   1:  PR[GP1:91,3] = PR[GP1:90,3] + 60.500;
   1:L PR[91] 10mm/sec CNT100;
   1:  PR[GP1:91,1] = PR[GP1:90,1] + -5.194;
   1:  PR[GP1:91,2] = PR[GP1:90,2] + -19.396;
   1:L PR[91] 10mm/sec CNT100;
   1:  PR[GP1:91,1] = PR[GP1:90,1] + -4.305;
   1:  PR[GP1:91,2] = PR[GP1:90,2] + -20.285;
   1:L PR[91] 10mm/sec CNT100;
   1:  PR[GP1:91,1] = PR[GP1:90,1] + -1.571;
   1:  PR[GP1:91,2] = PR[GP1:90,2] + -23.234;
   1:L PR[91] 10mm/sec CNT100;
   1:  PR[GP1:91,1] = PR[GP1:90,1] + -0.513;
   1:  PR[GP1:91,2] = PR[GP1:90,2] + -24.061;
   1:L PR[91] 10mm/sec CNT100;
   1:  PR[GP1:91,1] = PR[GP1:90,1] + 2.835;
   1:  PR[GP1:91,2] = PR[GP1:90,2] + -26.549;
   1:L PR[91] 10mm/sec CNT100;
   1:  PR[GP1:91,1] = PR[GP1:90,1] + 5.911;
   1:  PR[GP1:91,2] = PR[GP1:90,2] + -28.205;
   1:L PR[91] 10mm/sec CNT100;
   1:  PR[GP1:91,1] = PR[GP1:90,1] + 7.682;
   1:  PR[GP1:91,2] = PR[GP1:90,2] + -29.088;
   1:L PR[91] 10mm/sec CNT100;
   1:  PR[GP1:91,1] = PR[GP1:90,1] + 12.488;
   1:  PR[GP1:91,2] = PR[GP1:90,2] + -30.711;
   1:L PR[91] 10mm/sec CNT100;
   1:  PR[GP1:91,1] = PR[GP1:90,1] + 12.831;
   1:  PR[GP1:91,2] = PR[GP1:90,2] + -30.841;
   1:L PR[91] 10mm/sec CNT100;
   1:  PR[GP1:91,1] = PR[GP1:90,1] + 18.234;
   1:  PR[GP1:91,2] = PR[GP1:90,2] + -31.928;
   1:L PR[91] 10mm/sec CNT100;
   1:  PR[GP1:91,1] = PR[GP1:90,1] + 19.560;
   1:  PR[GP1:91,2] = PR[GP1:90,2] + -32.004;
   1:L PR[91] 10mm/sec CNT100;
   1:  PR[GP1:91,1] = PR[GP1:90,1] + 22.620;
   1:  PR[GP1:91,2] = PR[GP1:90,2] + -32.037;
   1:L PR[91] 10mm/sec CNT100;
   1:  PR[GP1:91,1] = PR[GP1:90,1] + 24.592;
   1:  PR[GP1:91,2] = PR[GP1:90,2] + -31.874;
   1:L PR[91] 10mm/sec CNT100;
   1:  PR[GP1:91,1] = PR[GP1:90,1] + 25.073;
   1:  PR[GP1:91,2] = PR[GP1:90,2] + -31.805;
   1:L PR[91] 10mm/sec CNT100;
   1:  PR[GP1:91,1] = PR[GP1:90,1] + 25.618;
   1:  PR[GP1:91,2] = PR[GP1:90,2] + -31.695;
   1:L PR[91] 10mm/sec CNT100;
   1:  PR[GP1:91,1] = PR[GP1:90,1] + 27.898;
   1:  PR[GP1:91,2] = PR[GP1:90,2] + -31.148;
   1:L PR[91] 10mm/sec CNT100;
   1:  PR[GP1:91,1] = PR[GP1:90,1] + 28.378;
   1:  PR[GP1:91,2] = PR[GP1:90,2] + -31.011;
   1:L PR[91] 10mm/sec CNT100;
   1:  PR[GP1:91,1] = PR[GP1:90,1] + 31.208;
   1:  PR[GP1:91,2] = PR[GP1:90,2] + -29.808;
   1:L PR[91] 10mm/sec CNT100;
   1:  PR[GP1:91,1] = PR[GP1:90,1] + 31.485;
   1:  PR[GP1:91,2] = PR[GP1:90,2] + -29.654;
   1:L PR[91] 10mm/sec CNT100;
   1:  PR[GP1:91,1] = PR[GP1:90,1] + 33.797;
   1:  PR[GP1:91,2] = PR[GP1:90,2] + -28.079;
   1:L PR[91] 10mm/sec CNT100;
   1:  PR[GP1:91,1] = PR[GP1:90,1] + 33.896;
   1:  PR[GP1:91,2] = PR[GP1:90,2] + -28.003;
   1:L PR[91] 10mm/sec CNT100;
   1:  PR[GP1:91,1] = PR[GP1:90,1] + 35.916;
   1:  PR[GP1:91,2] = PR[GP1:90,2] + -25.895;
   1:L PR[91] 10mm/sec CNT100;
   1:  PR[GP1:91,1] = PR[GP1:90,1] + 37.425;
   1:  PR[GP1:91,2] = PR[GP1:90,2] + -23.399;
   1:L PR[91] 10mm/sec CNT100;
   1:  PR[GP1:91,1] = PR[GP1:90,1] + 38.343;
   1:  PR[GP1:91,2] = PR[GP1:90,2] + -20.620;
   1:L PR[91] 10mm/sec CNT100;
   1:  PR[GP1:91,1] = PR[GP1:90,1] + 38.648;
   1:  PR[GP1:91,2] = PR[GP1:90,2] + -17.822;
   1:L PR[91] 10mm/sec CNT100;
   1:  PR[GP1:91,1] = PR[GP1:90,1] + 38.658;
   1:  PR[GP1:91,2] = PR[GP1:90,2] + -17.576;
   1:L PR[91] 10mm/sec CNT100;
   1:  PR[GP1:91,1] = PR[GP1:90,1] + 38.397;
   1:  PR[GP1:91,2] = PR[GP1:90,2] + -14.692;
   1:L PR[91] 10mm/sec CNT100;
   1:  PR[GP1:91,1] = PR[GP1:90,1] + 38.333;
   1:  PR[GP1:91,2] = PR[GP1:90,2] + -14.338;
   1:L PR[91] 10mm/sec CNT100;
   1:  PR[GP1:91,1] = PR[GP1:90,1] + 38.245;
   1:  PR[GP1:91,2] = PR[GP1:90,2] + -13.997;
   1:L PR[91] 10mm/sec CNT100;
   1:  PR[GP1:91,1] = PR[GP1:90,1] + 37.589;
   1:  PR[GP1:91,2] = PR[GP1:90,2] + -11.656;
   1:L PR[91] 10mm/sec CNT100;
   1:  PR[GP1:91,1] = PR[GP1:90,1] + 37.155;
   1:  PR[GP1:91,2] = PR[GP1:90,2] + -10.549;
   1:L PR[91] 10mm/sec CNT100;
   1:  PR[GP1:91,1] = PR[GP1:90,1] + 36.548;
   1:  PR[GP1:91,2] = PR[GP1:90,2] + -9.179;
   1:L PR[91] 10mm/sec CNT100;
   1:  PR[GP1:91,1] = PR[GP1:90,1] + 36.145;
   1:  PR[GP1:91,2] = PR[GP1:90,2] + -8.389;
   1:L PR[91] 10mm/sec CNT100;
   1:  PR[GP1:91,1] = PR[GP1:90,1] + 34.970;
   1:  PR[GP1:91,2] = PR[GP1:90,2] + -6.423;
   1:L PR[91] 10mm/sec CNT100;
   1:  PR[GP1:91,1] = PR[GP1:90,1] + 34.010;
   1:  PR[GP1:91,2] = PR[GP1:90,2] + -5.069;
   1:L PR[91] 10mm/sec CNT100;
   1:  PR[GP1:91,1] = PR[GP1:90,1] + 33.678;
   1:  PR[GP1:91,2] = PR[GP1:90,2] + -4.630;
   1:L PR[91] 10mm/sec CNT100;
   1:  PR[GP1:91,1] = PR[GP1:90,1] + 32.304;
   1:  PR[GP1:91,2] = PR[GP1:90,2] + -2.989;
   1:L PR[91] 10mm/sec CNT100;
   1:  PR[GP1:91,1] = PR[GP1:90,1] + 31.898;
   1:  PR[GP1:91,2] = PR[GP1:90,2] + -2.568;
   1:L PR[91] 10mm/sec CNT100;
   1:  PR[GP1:91,1] = PR[GP1:90,1] + 31.801;
   1:  PR[GP1:91,2] = PR[GP1:90,2] + -2.634;
   1:L PR[91] 10mm/sec CNT100;
   1:  PR[GP1:91,1] = PR[GP1:90,1] + 30.640;
   1:  PR[GP1:91,2] = PR[GP1:90,2] + -1.147;
   1:L PR[91] 10mm/sec CNT100;
   1:  PR[GP1:91,1] = PR[GP1:90,1] + 30.003;
   1:  PR[GP1:91,2] = PR[GP1:90,2] + -0.535;
   1:L PR[91] 10mm/sec CNT100;
   1:  PR[GP1:91,1] = PR[GP1:90,1] + 29.805;
   1:  PR[GP1:91,2] = PR[GP1:90,2] + -0.397;
   1:L PR[91] 10mm/sec CNT100;
   1:  PR[GP1:91,1] = PR[GP1:90,1] + 29.023;
   1:  PR[GP1:91,2] = PR[GP1:90,2] + 0.338;
   1:L PR[91] 10mm/sec CNT100;
   1:  PR[GP1:91,1] = PR[GP1:90,1] + 28.284;
   1:  PR[GP1:91,2] = PR[GP1:90,2] + 1.041;
   1:L PR[91] 10mm/sec CNT100;
   1:  PR[GP1:91,1] = PR[GP1:90,1] + 27.524;
   1:  PR[GP1:91,2] = PR[GP1:90,2] + 1.795;
   1:L PR[91] 10mm/sec CNT100;
   1:  PR[GP1:91,1] = PR[GP1:90,1] + 26.740;
   1:  PR[GP1:91,2] = PR[GP1:90,2] + 2.333;
   1:L PR[91] 10mm/sec CNT100;
   1:  PR[GP1:91,1] = PR[GP1:90,1] + 25.814;
   1:  PR[GP1:91,2] = PR[GP1:90,2] + 2.997;
   1:L PR[91] 10mm/sec CNT100;
   1:  PR[GP1:91,1] = PR[GP1:90,1] + 24.164;
   1:  PR[GP1:91,2] = PR[GP1:90,2] + 4.208;
   1:L PR[91] 10mm/sec CNT100;
   1:  PR[GP1:91,1] = PR[GP1:90,1] + 22.827;
   1:  PR[GP1:91,2] = PR[GP1:90,2] + 4.879;
   1:L PR[91] 10mm/sec CNT100;
   1:  PR[GP1:91,1] = PR[GP1:90,1] + 20.554;
   1:  PR[GP1:91,2] = PR[GP1:90,2] + 6.052;
   1:L PR[91] 10mm/sec CNT100;
   1:  PR[GP1:91,1] = PR[GP1:90,1] + 16.810;
   1:  PR[GP1:91,2] = PR[GP1:90,2] + 7.249;
   1:L PR[91] 10mm/sec CNT100;
   1:  PR[GP1:91,1] = PR[GP1:90,1] + 13.045;
   1:  PR[GP1:91,2] = PR[GP1:90,2] + 7.739;
   1:L PR[91] 10mm/sec CNT100;
   1:  PR[GP1:91,1] = PR[GP1:90,1] + 10.462;
   1:  PR[GP1:91,2] = PR[GP1:90,2] + 7.653;
   1:L PR[91] 10mm/sec CNT100;
   1:  PR[GP1:91,1] = PR[GP1:90,1] + 8.879;
   1:  PR[GP1:91,2] = PR[GP1:90,2] + 7.617;
   1:L PR[91] 10mm/sec CNT100;
   1:  PR[GP1:91,1] = PR[GP1:90,1] + 6.437;
   1:  PR[GP1:91,2] = PR[GP1:90,2] + 7.516;
   1:L PR[91] 10mm/sec CNT100;
   1:  PR[GP1:91,1] = PR[GP1:90,1] + 3.454;
   1:  PR[GP1:91,2] = PR[GP1:90,2] + 7.049;
   1:L PR[91] 10mm/sec CNT100;
   1:  PR[GP1:91,1] = PR[GP1:90,1] + 2.394;
   1:  PR[GP1:91,2] = PR[GP1:90,2] + 6.836;
   1:L PR[91] 10mm/sec CNT100;
   1:  PR[GP1:91,1] = PR[GP1:90,1] + -1.224;
   1:  PR[GP1:91,2] = PR[GP1:90,2] + 5.513;
   1:L PR[91] 10mm/sec CNT100;
   1:  PR[GP1:91,1] = PR[GP1:90,1] + -1.466;
   1:  PR[GP1:91,2] = PR[GP1:90,2] + 5.415;
   1:L PR[91] 10mm/sec CNT100;
   1:  PR[GP1:91,1] = PR[GP1:90,1] + -4.753;
   1:  PR[GP1:91,2] = PR[GP1:90,2] + 3.285;
   1:L PR[91] 10mm/sec CNT100;
   1:  PR[GP1:91,1] = PR[GP1:90,1] + -6.987;
   1:  PR[GP1:91,2] = PR[GP1:90,2] + 0.860;
   1:L PR[91] 10mm/sec CNT100;
   1:  PR[GP1:91,1] = PR[GP1:90,1] + -7.303;
   1:  PR[GP1:91,2] = PR[GP1:90,2] + 0.540;
   1:L PR[91] 10mm/sec CNT100;
   1:  PR[GP1:91,1] = PR[GP1:90,1] + -8.731;
   1:  PR[GP1:91,2] = PR[GP1:90,2] + -2.182;
   1:L PR[91] 10mm/sec CNT100;
   1:  PR[GP1:91,1] = PR[GP1:90,1] + -9.012;
   1:  PR[GP1:91,2] = PR[GP1:90,2] + -2.672;
   1:L PR[91] 10mm/sec CNT100;
   1:  PR[GP1:91,1] = PR[GP1:90,1] + -9.724;
   1:  PR[GP1:91,2] = PR[GP1:90,2] + -5.754;
   1:L PR[91] 10mm/sec CNT100;
   1:  PR[GP1:91,1] = PR[GP1:90,1] + -9.855;
   1:  PR[GP1:91,2] = PR[GP1:90,2] + -6.227;
   1:L PR[91] 10mm/sec CNT100;
   1:  PR[GP1:91,1] = PR[GP1:90,1] + -9.843;
   1:  PR[GP1:91,2] = PR[GP1:90,2] + -6.670;
   1:L PR[91] 10mm/sec CNT100;
   1:  PR[GP1:91,1] = PR[GP1:90,1] + -9.814;
   1:  PR[GP1:91,2] = PR[GP1:90,2] + -7.085;
   1:L PR[91] 10mm/sec CNT100;
   1:  PR[GP1:91,1] = PR[GP1:90,1] + -9.633;
   1:  PR[GP1:91,2] = PR[GP1:90,2] + -10.040;
   1:L PR[91] 10mm/sec CNT100;
   1:  PR[GP1:91,1] = PR[GP1:90,1] + -9.142;
   1:  PR[GP1:91,2] = PR[GP1:90,2] + -11.869;
   1:L PR[91] 10mm/sec CNT100;
   1:  PR[GP1:91,1] = PR[GP1:90,1] + -8.151;
   1:  PR[GP1:91,2] = PR[GP1:90,2] + -14.733;
   1:L PR[91] 10mm/sec CNT100;
   1:  PR[GP1:91,1] = PR[GP1:90,1] + -7.574;
   1:  PR[GP1:91,2] = PR[GP1:90,2] + -15.755;
   1:L PR[91] 10mm/sec CNT100;
   1:  PR[GP1:91,1] = PR[GP1:90,1] + -6.899;
   1:  PR[GP1:91,2] = PR[GP1:90,2] + -15.803;
   1:  PR[GP1:91,3] = PR[GP1:90,3] + 61.600;
   1:L PR[91] 10mm/sec CNT100;
   1:  PR[GP1:91,1] = PR[GP1:90,1] + -4.902;
   1:  PR[GP1:91,2] = PR[GP1:90,2] + -18.924;
   1:L PR[91] 10mm/sec CNT100;
   1:  PR[GP1:91,1] = PR[GP1:90,1] + -4.524;
   1:  PR[GP1:91,2] = PR[GP1:90,2] + -19.558;
   1:L PR[91] 10mm/sec CNT100;
   1:  PR[GP1:91,1] = PR[GP1:90,1] + -4.376;
   1:  PR[GP1:91,2] = PR[GP1:90,2] + -19.764;
   1:L PR[91] 10mm/sec CNT100;
   1:  PR[GP1:91,1] = PR[GP1:90,1] + -1.185;
   1:  PR[GP1:91,2] = PR[GP1:90,2] + -23.222;
   1:L PR[91] 10mm/sec CNT100;
   1:  PR[GP1:91,1] = PR[GP1:90,1] + -0.777;
   1:  PR[GP1:91,2] = PR[GP1:90,2] + -23.644;
   1:L PR[91] 10mm/sec CNT100;
   1:  PR[GP1:91,1] = PR[GP1:90,1] + 0.913;
   1:  PR[GP1:91,2] = PR[GP1:90,2] + -24.966;
   1:L PR[91] 10mm/sec CNT100;
   1:  PR[GP1:91,1] = PR[GP1:90,1] + 3.607;
   1:  PR[GP1:91,2] = PR[GP1:90,2] + -26.967;
   1:L PR[91] 10mm/sec CNT100;
   1:  PR[GP1:91,1] = PR[GP1:90,1] + 7.393;
   1:  PR[GP1:91,2] = PR[GP1:90,2] + -29.006;
   1:L PR[91] 10mm/sec CNT100;
   1:  PR[GP1:91,1] = PR[GP1:90,1] + 8.431;
   1:  PR[GP1:91,2] = PR[GP1:90,2] + -29.523;
   1:L PR[91] 10mm/sec CNT100;
   1:  PR[GP1:91,1] = PR[GP1:90,1] + 11.289;
   1:  PR[GP1:91,2] = PR[GP1:90,2] + -30.488;
   1:L PR[91] 10mm/sec CNT100;
   1:  PR[GP1:91,1] = PR[GP1:90,1] + 13.911;
   1:  PR[GP1:91,2] = PR[GP1:90,2] + -31.485;
   1:L PR[91] 10mm/sec CNT100;
   1:  PR[GP1:91,1] = PR[GP1:90,1] + 19.104;
   1:  PR[GP1:91,2] = PR[GP1:90,2] + -32.524;
   1:L PR[91] 10mm/sec CNT100;
   1:  PR[GP1:91,1] = PR[GP1:90,1] + 20.959;
   1:  PR[GP1:91,2] = PR[GP1:90,2] + -32.631;
   1:L PR[91] 10mm/sec CNT100;
   1:  PR[GP1:91,1] = PR[GP1:90,1] + 23.332;
   1:  PR[GP1:91,2] = PR[GP1:90,2] + -32.657;
   1:L PR[91] 10mm/sec CNT100;
   1:  PR[GP1:91,1] = PR[GP1:90,1] + 25.733;
   1:  PR[GP1:91,2] = PR[GP1:90,2] + -32.458;
   1:L PR[91] 10mm/sec CNT100;
   1:  PR[GP1:91,1] = PR[GP1:90,1] + 26.050;
   1:  PR[GP1:91,2] = PR[GP1:90,2] + -32.413;
   1:L PR[91] 10mm/sec CNT100;
   1:  PR[GP1:91,1] = PR[GP1:90,1] + 26.413;
   1:  PR[GP1:91,2] = PR[GP1:90,2] + -32.339;
   1:L PR[91] 10mm/sec CNT100;
   1:  PR[GP1:91,1] = PR[GP1:90,1] + 29.153;
   1:  PR[GP1:91,2] = PR[GP1:90,2] + -31.681;
   1:L PR[91] 10mm/sec CNT100;
   1:  PR[GP1:91,1] = PR[GP1:90,1] + 29.369;
   1:  PR[GP1:91,2] = PR[GP1:90,2] + -31.620;
   1:L PR[91] 10mm/sec CNT100;
   1:  PR[GP1:91,1] = PR[GP1:90,1] + 32.379;
   1:  PR[GP1:91,2] = PR[GP1:90,2] + -30.326;
   1:L PR[91] 10mm/sec CNT100;
   1:  PR[GP1:91,1] = PR[GP1:90,1] + 32.945;
   1:  PR[GP1:91,2] = PR[GP1:90,2] + -29.940;
   1:L PR[91] 10mm/sec CNT100;
   1:  PR[GP1:91,1] = PR[GP1:90,1] + 34.716;
   1:  PR[GP1:91,2] = PR[GP1:90,2] + -28.678;
   1:L PR[91] 10mm/sec CNT100;
   1:  PR[GP1:91,1] = PR[GP1:90,1] + 34.917;
   1:  PR[GP1:91,2] = PR[GP1:90,2] + -28.521;
   1:L PR[91] 10mm/sec CNT100;
   1:  PR[GP1:91,1] = PR[GP1:90,1] + 36.783;
   1:  PR[GP1:91,2] = PR[GP1:90,2] + -26.529;
   1:L PR[91] 10mm/sec CNT100;
   1:  PR[GP1:91,1] = PR[GP1:90,1] + 37.004;
   1:  PR[GP1:91,2] = PR[GP1:90,2] + -26.199;
   1:L PR[91] 10mm/sec CNT100;
   1:  PR[GP1:91,1] = PR[GP1:90,1] + 38.367;
   1:  PR[GP1:91,2] = PR[GP1:90,2] + -23.935;
   1:L PR[91] 10mm/sec CNT100;
   1:  PR[GP1:91,1] = PR[GP1:90,1] + 39.330;
   1:  PR[GP1:91,2] = PR[GP1:90,2] + -21.121;
   1:L PR[91] 10mm/sec CNT100;
   1:  PR[GP1:91,1] = PR[GP1:90,1] + 39.707;
   1:  PR[GP1:91,2] = PR[GP1:90,2] + -18.156;
   1:L PR[91] 10mm/sec CNT100;
   1:  PR[GP1:91,1] = PR[GP1:90,1] + 39.704;
   1:  PR[GP1:91,2] = PR[GP1:90,2] + -18.109;
   1:L PR[91] 10mm/sec CNT100;
   1:  PR[GP1:91,1] = PR[GP1:90,1] + 39.428;
   1:  PR[GP1:91,2] = PR[GP1:90,2] + -15.086;
   1:L PR[91] 10mm/sec CNT100;
   1:  PR[GP1:91,1] = PR[GP1:90,1] + 39.406;
   1:  PR[GP1:91,2] = PR[GP1:90,2] + -14.965;
   1:L PR[91] 10mm/sec CNT100;
   1:  PR[GP1:91,1] = PR[GP1:90,1] + 38.590;
   1:  PR[GP1:91,2] = PR[GP1:90,2] + -12.026;
   1:L PR[91] 10mm/sec CNT100;
   1:  PR[GP1:91,1] = PR[GP1:90,1] + 38.315;
   1:  PR[GP1:91,2] = PR[GP1:90,2] + -11.324;
   1:L PR[91] 10mm/sec CNT100;
   1:  PR[GP1:91,1] = PR[GP1:90,1] + 37.525;
   1:  PR[GP1:91,2] = PR[GP1:90,2] + -9.542;
   1:L PR[91] 10mm/sec CNT100;
   1:  PR[GP1:91,1] = PR[GP1:90,1] + 37.230;
   1:  PR[GP1:91,2] = PR[GP1:90,2] + -8.964;
   1:L PR[91] 10mm/sec CNT100;
   1:  PR[GP1:91,1] = PR[GP1:90,1] + 35.968;
   1:  PR[GP1:91,2] = PR[GP1:90,2] + -6.849;
   1:L PR[91] 10mm/sec CNT100;
   1:  PR[GP1:91,1] = PR[GP1:90,1] + 35.201;
   1:  PR[GP1:91,2] = PR[GP1:90,2] + -5.768;
   1:L PR[91] 10mm/sec CNT100;
   1:  PR[GP1:91,1] = PR[GP1:90,1] + 34.586;
   1:  PR[GP1:91,2] = PR[GP1:90,2] + -4.954;
   1:L PR[91] 10mm/sec CNT100;
   1:  PR[GP1:91,1] = PR[GP1:90,1] + 33.428;
   1:  PR[GP1:91,2] = PR[GP1:90,2] + -3.571;
   1:L PR[91] 10mm/sec CNT100;
   1:  PR[GP1:91,1] = PR[GP1:90,1] + 33.059;
   1:  PR[GP1:91,2] = PR[GP1:90,2] + -3.175;
   1:L PR[91] 10mm/sec CNT100;
   1:  PR[GP1:91,1] = PR[GP1:90,1] + 31.368;
   1:  PR[GP1:91,2] = PR[GP1:90,2] + -1.469;
   1:L PR[91] 10mm/sec CNT100;
   1:  PR[GP1:91,1] = PR[GP1:90,1] + 30.956;
   1:  PR[GP1:91,2] = PR[GP1:90,2] + -1.099;
   1:L PR[91] 10mm/sec CNT100;
   1:  PR[GP1:91,1] = PR[GP1:90,1] + 30.907;
   1:  PR[GP1:91,2] = PR[GP1:90,2] + -1.075;
   1:L PR[91] 10mm/sec CNT100;
   1:  PR[GP1:91,1] = PR[GP1:90,1] + 30.645;
   1:  PR[GP1:91,2] = PR[GP1:90,2] + -0.856;
   1:L PR[91] 10mm/sec CNT100;
   1:  PR[GP1:91,1] = PR[GP1:90,1] + 29.919;
   1:  PR[GP1:91,2] = PR[GP1:90,2] + -0.156;
   1:L PR[91] 10mm/sec CNT100;
   1:  PR[GP1:91,1] = PR[GP1:90,1] + 29.499;
   1:  PR[GP1:91,2] = PR[GP1:90,2] + 0.136;
   1:L PR[91] 10mm/sec CNT100;
   1:  PR[GP1:91,1] = PR[GP1:90,1] + 28.083;
   1:  PR[GP1:91,2] = PR[GP1:90,2] + 1.466;
   1:L PR[91] 10mm/sec CNT100;
   1:  PR[GP1:91,1] = PR[GP1:90,1] + 26.293;
   1:  PR[GP1:91,2] = PR[GP1:90,2] + 2.692;
   1:L PR[91] 10mm/sec CNT100;
   1:  PR[GP1:91,1] = PR[GP1:90,1] + 24.680;
   1:  PR[GP1:91,2] = PR[GP1:90,2] + 3.848;
   1:L PR[91] 10mm/sec CNT100;
   1:  PR[GP1:91,1] = PR[GP1:90,1] + 22.266;
   1:  PR[GP1:91,2] = PR[GP1:90,2] + 5.052;
   1:L PR[91] 10mm/sec CNT100;
   1:  PR[GP1:91,1] = PR[GP1:90,1] + 21.047;
   1:  PR[GP1:91,2] = PR[GP1:90,2] + 5.681;
   1:L PR[91] 10mm/sec CNT100;
   1:  PR[GP1:91,1] = PR[GP1:90,1] + 17.283;
   1:  PR[GP1:91,2] = PR[GP1:90,2] + 6.871;
   1:L PR[91] 10mm/sec CNT100;
   1:  PR[GP1:91,1] = PR[GP1:90,1] + 13.493;
   1:  PR[GP1:91,2] = PR[GP1:90,2] + 7.364;
   1:L PR[91] 10mm/sec CNT100;
   1:  PR[GP1:91,1] = PR[GP1:90,1] + 12.502;
   1:  PR[GP1:91,2] = PR[GP1:90,2] + 7.353;
   1:L PR[91] 10mm/sec CNT100;
   1:  PR[GP1:91,1] = PR[GP1:90,1] + 10.236;
   1:  PR[GP1:91,2] = PR[GP1:90,2] + 7.289;
   1:L PR[91] 10mm/sec CNT100;
   1:  PR[GP1:91,1] = PR[GP1:90,1] + 7.160;
   1:  PR[GP1:91,2] = PR[GP1:90,2] + 7.162;
   1:L PR[91] 10mm/sec CNT100;
   1:  PR[GP1:91,1] = PR[GP1:90,1] + 4.784;
   1:  PR[GP1:91,2] = PR[GP1:90,2] + 6.790;
   1:L PR[91] 10mm/sec CNT100;
   1:  PR[GP1:91,1] = PR[GP1:90,1] + 3.183;
   1:  PR[GP1:91,2] = PR[GP1:90,2] + 6.469;
   1:L PR[91] 10mm/sec CNT100;
   1:  PR[GP1:91,1] = PR[GP1:90,1] + 0.123;
   1:  PR[GP1:91,2] = PR[GP1:90,2] + 5.350;
   1:L PR[91] 10mm/sec CNT100;
   1:  PR[GP1:91,1] = PR[GP1:90,1] + -0.614;
   1:  PR[GP1:91,2] = PR[GP1:90,2] + 5.061;
   1:L PR[91] 10mm/sec CNT100;
   1:  PR[GP1:91,1] = PR[GP1:90,1] + -0.655;
   1:  PR[GP1:91,2] = PR[GP1:90,2] + 5.040;
   1:L PR[91] 10mm/sec CNT100;
   1:  PR[GP1:91,1] = PR[GP1:90,1] + -3.900;
   1:  PR[GP1:91,2] = PR[GP1:90,2] + 2.951;
   1:L PR[91] 10mm/sec CNT100;
   1:  PR[GP1:91,1] = PR[GP1:90,1] + -3.952;
   1:  PR[GP1:91,2] = PR[GP1:90,2] + 2.906;
   1:L PR[91] 10mm/sec CNT100;
   1:  PR[GP1:91,1] = PR[GP1:90,1] + -6.462;
   1:  PR[GP1:91,2] = PR[GP1:90,2] + 0.194;
   1:L PR[91] 10mm/sec CNT100;
   1:  PR[GP1:91,1] = PR[GP1:90,1] + -8.163;
   1:  PR[GP1:91,2] = PR[GP1:90,2] + -3.034;
   1:L PR[91] 10mm/sec CNT100;
   1:  PR[GP1:91,1] = PR[GP1:90,1] + -8.990;
   1:  PR[GP1:91,2] = PR[GP1:90,2] + -6.594;
   1:L PR[91] 10mm/sec CNT100;
   1:  PR[GP1:91,1] = PR[GP1:90,1] + -8.943;
   1:  PR[GP1:91,2] = PR[GP1:90,2] + -7.401;
   1:L PR[91] 10mm/sec CNT100;
   1:  PR[GP1:91,1] = PR[GP1:90,1] + -8.788;
   1:  PR[GP1:91,2] = PR[GP1:90,2] + -10.327;
   1:L PR[91] 10mm/sec CNT100;
   1:  PR[GP1:91,1] = PR[GP1:90,1] + -8.767;
   1:  PR[GP1:91,2] = PR[GP1:90,2] + -10.461;
   1:L PR[91] 10mm/sec CNT100;
   1:  PR[GP1:91,1] = PR[GP1:90,1] + -8.391;
   1:  PR[GP1:91,2] = PR[GP1:90,2] + -11.876;
   1:L PR[91] 10mm/sec CNT100;
   1:  PR[GP1:91,1] = PR[GP1:90,1] + -7.244;
   1:  PR[GP1:91,2] = PR[GP1:90,2] + -15.190;
   1:L PR[91] 10mm/sec CNT100;
   1:  PR[GP1:91,1] = PR[GP1:90,1] + -6.223;
   1:  PR[GP1:91,2] = PR[GP1:90,2] + -15.851;
   1:  PR[GP1:91,3] = PR[GP1:90,3] + 62.700;
   1:L PR[91] 10mm/sec CNT100;
   1:  PR[GP1:91,1] = PR[GP1:90,1] + -5.431;
   1:  PR[GP1:91,2] = PR[GP1:90,2] + -17.089;
   1:L PR[91] 10mm/sec CNT100;
   1:  PR[GP1:91,1] = PR[GP1:90,1] + -3.948;
   1:  PR[GP1:91,2] = PR[GP1:90,2] + -19.575;
   1:L PR[91] 10mm/sec CNT100;
   1:  PR[GP1:91,1] = PR[GP1:90,1] + -3.262;
   1:  PR[GP1:91,2] = PR[GP1:90,2] + -20.527;
   1:L PR[91] 10mm/sec CNT100;
   1:  PR[GP1:91,1] = PR[GP1:90,1] + -0.547;
   1:  PR[GP1:91,2] = PR[GP1:90,2] + -23.470;
   1:L PR[91] 10mm/sec CNT100;
   1:  PR[GP1:91,1] = PR[GP1:90,1] + 0.021;
   1:  PR[GP1:91,2] = PR[GP1:90,2] + -24.057;
   1:L PR[91] 10mm/sec CNT100;
   1:  PR[GP1:91,1] = PR[GP1:90,1] + 2.339;
   1:  PR[GP1:91,2] = PR[GP1:90,2] + -25.870;
   1:L PR[91] 10mm/sec CNT100;
   1:  PR[GP1:91,1] = PR[GP1:90,1] + 4.380;
   1:  PR[GP1:91,2] = PR[GP1:90,2] + -27.386;
   1:L PR[91] 10mm/sec CNT100;
   1:  PR[GP1:91,1] = PR[GP1:90,1] + 8.875;
   1:  PR[GP1:91,2] = PR[GP1:90,2] + -29.807;
   1:L PR[91] 10mm/sec CNT100;
   1:  PR[GP1:91,1] = PR[GP1:90,1] + 9.179;
   1:  PR[GP1:91,2] = PR[GP1:90,2] + -29.959;
   1:L PR[91] 10mm/sec CNT100;
   1:  PR[GP1:91,1] = PR[GP1:90,1] + 10.090;
   1:  PR[GP1:91,2] = PR[GP1:90,2] + -30.266;
   1:L PR[91] 10mm/sec CNT100;
   1:  PR[GP1:91,1] = PR[GP1:90,1] + 14.991;
   1:  PR[GP1:91,2] = PR[GP1:90,2] + -32.128;
   1:L PR[91] 10mm/sec CNT100;
   1:  PR[GP1:91,1] = PR[GP1:90,1] + 19.975;
   1:  PR[GP1:91,2] = PR[GP1:90,2] + -33.121;
   1:L PR[91] 10mm/sec CNT100;
   1:  PR[GP1:91,1] = PR[GP1:90,1] + 22.358;
   1:  PR[GP1:91,2] = PR[GP1:90,2] + -33.258;
   1:L PR[91] 10mm/sec CNT100;
   1:  PR[GP1:91,1] = PR[GP1:90,1] + 24.044;
   1:  PR[GP1:91,2] = PR[GP1:90,2] + -33.276;
   1:L PR[91] 10mm/sec CNT100;
   1:  PR[GP1:91,1] = PR[GP1:90,1] + 26.863;
   1:  PR[GP1:91,2] = PR[GP1:90,2] + -33.043;
   1:L PR[91] 10mm/sec CNT100;
   1:  PR[GP1:91,1] = PR[GP1:90,1] + 27.217;
   1:  PR[GP1:91,2] = PR[GP1:90,2] + -32.982;
   1:L PR[91] 10mm/sec CNT100;
   1:  PR[GP1:91,1] = PR[GP1:90,1] + 30.366;
   1:  PR[GP1:91,2] = PR[GP1:90,2] + -32.225;
   1:L PR[91] 10mm/sec CNT100;
   1:  PR[GP1:91,1] = PR[GP1:90,1] + 33.261;
   1:  PR[GP1:91,2] = PR[GP1:90,2] + -30.893;
   1:L PR[91] 10mm/sec CNT100;
   1:  PR[GP1:91,1] = PR[GP1:90,1] + 35.260;
   1:  PR[GP1:91,2] = PR[GP1:90,2] + -29.468;
   1:L PR[91] 10mm/sec CNT100;
   1:  PR[GP1:91,1] = PR[GP1:90,1] + 36.005;
   1:  PR[GP1:91,2] = PR[GP1:90,2] + -28.884;
   1:L PR[91] 10mm/sec CNT100;
   1:  PR[GP1:91,1] = PR[GP1:90,1] + 37.585;
   1:  PR[GP1:91,2] = PR[GP1:90,2] + -27.197;
   1:L PR[91] 10mm/sec CNT100;
   1:  PR[GP1:91,1] = PR[GP1:90,1] + 38.135;
   1:  PR[GP1:91,2] = PR[GP1:90,2] + -26.377;
   1:L PR[91] 10mm/sec CNT100;
   1:  PR[GP1:91,1] = PR[GP1:90,1] + 39.289;
   1:  PR[GP1:91,2] = PR[GP1:90,2] + -24.459;
   1:L PR[91] 10mm/sec CNT100;
   1:  PR[GP1:91,1] = PR[GP1:90,1] + 40.268;
   1:  PR[GP1:91,2] = PR[GP1:90,2] + -21.575;
   1:L PR[91] 10mm/sec CNT100;
   1:  PR[GP1:91,1] = PR[GP1:90,1] + 40.593;
   1:  PR[GP1:91,2] = PR[GP1:90,2] + -19.026;
   1:L PR[91] 10mm/sec CNT100;
   1:  PR[GP1:91,1] = PR[GP1:90,1] + 40.632;
   1:  PR[GP1:91,2] = PR[GP1:90,2] + -18.615;
   1:L PR[91] 10mm/sec CNT100;
   1:  PR[GP1:91,1] = PR[GP1:90,1] + 40.433;
   1:  PR[GP1:91,2] = PR[GP1:90,2] + -15.506;
   1:L PR[91] 10mm/sec CNT100;
   1:  PR[GP1:91,1] = PR[GP1:90,1] + 40.290;
   1:  PR[GP1:91,2] = PR[GP1:90,2] + -14.910;
   1:L PR[91] 10mm/sec CNT100;
   1:  PR[GP1:91,1] = PR[GP1:90,1] + 39.592;
   1:  PR[GP1:91,2] = PR[GP1:90,2] + -12.397;
   1:L PR[91] 10mm/sec CNT100;
   1:  PR[GP1:91,1] = PR[GP1:90,1] + 39.475;
   1:  PR[GP1:91,2] = PR[GP1:90,2] + -12.098;
   1:L PR[91] 10mm/sec CNT100;
   1:  PR[GP1:91,1] = PR[GP1:90,1] + 38.503;
   1:  PR[GP1:91,2] = PR[GP1:90,2] + -9.905;
   1:L PR[91] 10mm/sec CNT100;
   1:  PR[GP1:91,1] = PR[GP1:90,1] + 38.316;
   1:  PR[GP1:91,2] = PR[GP1:90,2] + -9.538;
   1:L PR[91] 10mm/sec CNT100;
   1:  PR[GP1:91,1] = PR[GP1:90,1] + 36.965;
   1:  PR[GP1:91,2] = PR[GP1:90,2] + -7.276;
   1:L PR[91] 10mm/sec CNT100;
   1:  PR[GP1:91,1] = PR[GP1:90,1] + 36.391;
   1:  PR[GP1:91,2] = PR[GP1:90,2] + -6.467;
   1:L PR[91] 10mm/sec CNT100;
   1:  PR[GP1:91,1] = PR[GP1:90,1] + 35.494;
   1:  PR[GP1:91,2] = PR[GP1:90,2] + -5.279;
   1:L PR[91] 10mm/sec CNT100;
   1:  PR[GP1:91,1] = PR[GP1:90,1] + 34.556;
   1:  PR[GP1:91,2] = PR[GP1:90,2] + -4.158;
   1:L PR[91] 10mm/sec CNT100;
   1:  PR[GP1:91,1] = PR[GP1:90,1] + 33.888;
   1:  PR[GP1:91,2] = PR[GP1:90,2] + -3.442;
   1:L PR[91] 10mm/sec CNT100;
   1:  PR[GP1:91,1] = PR[GP1:90,1] + 32.451;
   1:  PR[GP1:91,2] = PR[GP1:90,2] + -1.992;
   1:L PR[91] 10mm/sec CNT100;
   1:  PR[GP1:91,1] = PR[GP1:90,1] + 31.380;
   1:  PR[GP1:91,2] = PR[GP1:90,2] + -1.036;
   1:L PR[91] 10mm/sec CNT100;
   1:  PR[GP1:91,1] = PR[GP1:90,1] + 29.989;
   1:  PR[GP1:91,2] = PR[GP1:90,2] + -0.003;
   1:L PR[91] 10mm/sec CNT100;
   1:  PR[GP1:91,1] = PR[GP1:90,1] + 29.851;
   1:  PR[GP1:91,2] = PR[GP1:90,2] + 0.196;
   1:L PR[91] 10mm/sec CNT100;
   1:  PR[GP1:91,1] = PR[GP1:90,1] + 29.189;
   1:  PR[GP1:91,2] = PR[GP1:90,2] + 0.672;
   1:L PR[91] 10mm/sec CNT100;
   1:  PR[GP1:91,1] = PR[GP1:90,1] + 28.661;
   1:  PR[GP1:91,2] = PR[GP1:90,2] + 1.168;
   1:L PR[91] 10mm/sec CNT100;
   1:  PR[GP1:91,1] = PR[GP1:90,1] + 28.057;
   1:  PR[GP1:91,2] = PR[GP1:90,2] + 1.598;
   1:L PR[91] 10mm/sec CNT100;
   1:  PR[GP1:91,1] = PR[GP1:90,1] + 27.643;
   1:  PR[GP1:91,2] = PR[GP1:90,2] + 1.819;
   1:L PR[91] 10mm/sec CNT100;
   1:  PR[GP1:91,1] = PR[GP1:90,1] + 25.846;
   1:  PR[GP1:91,2] = PR[GP1:90,2] + 3.050;
   1:L PR[91] 10mm/sec CNT100;
   1:  PR[GP1:91,1] = PR[GP1:90,1] + 25.208;
   1:  PR[GP1:91,2] = PR[GP1:90,2] + 3.507;
   1:L PR[91] 10mm/sec CNT100;
   1:  PR[GP1:91,1] = PR[GP1:90,1] + 23.937;
   1:  PR[GP1:91,2] = PR[GP1:90,2] + 4.110;
   1:L PR[91] 10mm/sec CNT100;
   1:  PR[GP1:91,1] = PR[GP1:90,1] + 21.545;
   1:  PR[GP1:91,2] = PR[GP1:90,2] + 5.309;
   1:L PR[91] 10mm/sec CNT100;
   1:  PR[GP1:91,1] = PR[GP1:90,1] + 17.761;
   1:  PR[GP1:91,2] = PR[GP1:90,2] + 6.492;
   1:L PR[91] 10mm/sec CNT100;
   1:  PR[GP1:91,1] = PR[GP1:90,1] + 13.949;
   1:  PR[GP1:91,2] = PR[GP1:90,2] + 6.988;
   1:L PR[91] 10mm/sec CNT100;
   1:  PR[GP1:91,1] = PR[GP1:90,1] + 13.061;
   1:L PR[91] 10mm/sec CNT100;
   1:  PR[GP1:91,1] = PR[GP1:90,1] + 11.579;
   1:  PR[GP1:91,2] = PR[GP1:90,2] + 6.961;
   1:L PR[91] 10mm/sec CNT100;
   1:  PR[GP1:91,1] = PR[GP1:90,1] + 7.883;
   1:  PR[GP1:91,2] = PR[GP1:90,2] + 6.808;
   1:L PR[91] 10mm/sec CNT100;
   1:  PR[GP1:91,1] = PR[GP1:90,1] + 6.113;
   1:  PR[GP1:91,2] = PR[GP1:90,2] + 6.531;
   1:L PR[91] 10mm/sec CNT100;
   1:  PR[GP1:91,1] = PR[GP1:90,1] + 3.971;
   1:  PR[GP1:91,2] = PR[GP1:90,2] + 6.101;
   1:L PR[91] 10mm/sec CNT100;
   1:  PR[GP1:91,1] = PR[GP1:90,1] + 1.474;
   1:  PR[GP1:91,2] = PR[GP1:90,2] + 5.188;
   1:L PR[91] 10mm/sec CNT100;
   1:  PR[GP1:91,1] = PR[GP1:90,1] + 0.236;
   1:  PR[GP1:91,2] = PR[GP1:90,2] + 4.702;
   1:L PR[91] 10mm/sec CNT100;
   1:  PR[GP1:91,1] = PR[GP1:90,1] + 0.131;
   1:  PR[GP1:91,2] = PR[GP1:90,2] + 4.648;
   1:L PR[91] 10mm/sec CNT100;
   1:  PR[GP1:91,1] = PR[GP1:90,1] + -2.947;
   1:  PR[GP1:91,2] = PR[GP1:90,2] + 2.669;
   1:L PR[91] 10mm/sec CNT100;
   1:  PR[GP1:91,1] = PR[GP1:90,1] + -3.269;
   1:  PR[GP1:91,2] = PR[GP1:90,2] + 2.386;
   1:L PR[91] 10mm/sec CNT100;
   1:  PR[GP1:91,1] = PR[GP1:90,1] + -5.490;
   1:  PR[GP1:91,2] = PR[GP1:90,2] + -0.014;
   1:L PR[91] 10mm/sec CNT100;
   1:  PR[GP1:91,1] = PR[GP1:90,1] + -5.625;
   1:  PR[GP1:91,2] = PR[GP1:90,2] + -0.179;
   1:L PR[91] 10mm/sec CNT100;
   1:  PR[GP1:91,1] = PR[GP1:90,1] + -5.732;
   1:  PR[GP1:91,2] = PR[GP1:90,2] + -0.371;
   1:L PR[91] 10mm/sec CNT100;
   1:  PR[GP1:91,1] = PR[GP1:90,1] + -7.293;
   1:  PR[GP1:91,2] = PR[GP1:90,2] + -3.345;
   1:L PR[91] 10mm/sec CNT100;
   1:  PR[GP1:91,1] = PR[GP1:90,1] + -7.336;
   1:  PR[GP1:91,2] = PR[GP1:90,2] + -3.468;
   1:L PR[91] 10mm/sec CNT100;
   1:  PR[GP1:91,1] = PR[GP1:90,1] + -8.094;
   1:  PR[GP1:91,2] = PR[GP1:90,2] + -6.733;
   1:L PR[91] 10mm/sec CNT100;
   1:  PR[GP1:91,1] = PR[GP1:90,1] + -8.136;
   1:  PR[GP1:91,2] = PR[GP1:90,2] + -6.962;
   1:L PR[91] 10mm/sec CNT100;
   1:  PR[GP1:91,1] = PR[GP1:90,1] + -8.140;
   1:  PR[GP1:91,2] = PR[GP1:90,2] + -7.191;
   1:L PR[91] 10mm/sec CNT100;
   1:  PR[GP1:91,1] = PR[GP1:90,1] + -7.967;
   1:  PR[GP1:91,2] = PR[GP1:90,2] + -10.473;
   1:L PR[91] 10mm/sec CNT100;
   1:  PR[GP1:91,1] = PR[GP1:90,1] + -7.893;
   1:  PR[GP1:91,2] = PR[GP1:90,2] + -10.928;
   1:L PR[91] 10mm/sec CNT100;
   1:  PR[GP1:91,1] = PR[GP1:90,1] + -7.640;
   1:  PR[GP1:91,2] = PR[GP1:90,2] + -11.882;
   1:L PR[91] 10mm/sec CNT100;
   1:  PR[GP1:91,1] = PR[GP1:90,1] + -6.337;
   1:  PR[GP1:91,2] = PR[GP1:90,2] + -15.648;
   1:L PR[91] 10mm/sec CNT100;
   1:  PR[GP1:91,1] = PR[GP1:90,1] + -5.476;
   1:  PR[GP1:91,2] = PR[GP1:90,2] + -16.037;
   1:  PR[GP1:91,3] = PR[GP1:90,3] + 63.800;
   1:L PR[91] 10mm/sec CNT100;
   1:  PR[GP1:91,1] = PR[GP1:90,1] + -5.415;
   1:  PR[GP1:91,2] = PR[GP1:90,2] + -16.166;
   1:L PR[91] 10mm/sec CNT100;
   1:  PR[GP1:91,1] = PR[GP1:90,1] + -3.372;
   1:  PR[GP1:91,2] = PR[GP1:90,2] + -19.593;
   1:L PR[91] 10mm/sec CNT100;
   1:  PR[GP1:91,1] = PR[GP1:90,1] + -2.148;
   1:  PR[GP1:91,2] = PR[GP1:90,2] + -21.290;
   1:L PR[91] 10mm/sec CNT100;
   1:  PR[GP1:91,1] = PR[GP1:90,1] + 0.091;
   1:  PR[GP1:91,2] = PR[GP1:90,2] + -23.717;
   1:L PR[91] 10mm/sec CNT100;
   1:  PR[GP1:91,1] = PR[GP1:90,1] + 0.820;
   1:  PR[GP1:91,2] = PR[GP1:90,2] + -24.471;
   1:L PR[91] 10mm/sec CNT100;
   1:  PR[GP1:91,1] = PR[GP1:90,1] + 3.765;
   1:  PR[GP1:91,2] = PR[GP1:90,2] + -26.774;
   1:L PR[91] 10mm/sec CNT100;
   1:  PR[GP1:91,1] = PR[GP1:90,1] + 5.152;
   1:  PR[GP1:91,2] = PR[GP1:90,2] + -27.805;
   1:L PR[91] 10mm/sec CNT100;
   1:  PR[GP1:91,1] = PR[GP1:90,1] + 9.077;
   1:  PR[GP1:91,2] = PR[GP1:90,2] + -29.919;
   1:L PR[91] 10mm/sec CNT100;
   1:  PR[GP1:91,1] = PR[GP1:90,1] + 10.016;
   1:  PR[GP1:91,2] = PR[GP1:90,2] + -30.469;
   1:L PR[91] 10mm/sec CNT100;
   1:  PR[GP1:91,1] = PR[GP1:90,1] + 16.071;
   1:  PR[GP1:91,2] = PR[GP1:90,2] + -32.772;
   1:L PR[91] 10mm/sec CNT100;
   1:  PR[GP1:91,1] = PR[GP1:90,1] + 20.845;
   1:  PR[GP1:91,2] = PR[GP1:90,2] + -33.718;
   1:L PR[91] 10mm/sec CNT100;
   1:  PR[GP1:91,1] = PR[GP1:90,1] + 23.758;
   1:  PR[GP1:91,2] = PR[GP1:90,2] + -33.885;
   1:L PR[91] 10mm/sec CNT100;
   1:  PR[GP1:91,1] = PR[GP1:90,1] + 24.756;
   1:  PR[GP1:91,2] = PR[GP1:90,2] + -33.896;
   1:L PR[91] 10mm/sec CNT100;
   1:  PR[GP1:91,1] = PR[GP1:90,1] + 28.040;
   1:  PR[GP1:91,2] = PR[GP1:90,2] + -33.619;
   1:L PR[91] 10mm/sec CNT100;
   1:  PR[GP1:91,1] = PR[GP1:90,1] + 28.455;
   1:  PR[GP1:91,2] = PR[GP1:90,2] + -33.520;
   1:L PR[91] 10mm/sec CNT100;
   1:  PR[GP1:91,1] = PR[GP1:90,1] + 30.921;
   1:  PR[GP1:91,2] = PR[GP1:90,2] + -32.863;
   1:L PR[91] 10mm/sec CNT100;
   1:  PR[GP1:91,1] = PR[GP1:90,1] + 31.737;
   1:  PR[GP1:91,2] = PR[GP1:90,2] + -32.547;
   1:L PR[91] 10mm/sec CNT100;
   1:  PR[GP1:91,1] = PR[GP1:90,1] + 34.162;
   1:  PR[GP1:91,2] = PR[GP1:90,2] + -31.429;
   1:L PR[91] 10mm/sec CNT100;
   1:  PR[GP1:91,1] = PR[GP1:90,1] + 35.804;
   1:  PR[GP1:91,2] = PR[GP1:90,2] + -30.259;
   1:L PR[91] 10mm/sec CNT100;
   1:  PR[GP1:91,1] = PR[GP1:90,1] + 37.092;
   1:  PR[GP1:91,2] = PR[GP1:90,2] + -29.247;
   1:L PR[91] 10mm/sec CNT100;
   1:  PR[GP1:91,1] = PR[GP1:90,1] + 38.387;
   1:  PR[GP1:91,2] = PR[GP1:90,2] + -27.865;
   1:L PR[91] 10mm/sec CNT100;
   1:  PR[GP1:91,1] = PR[GP1:90,1] + 39.265;
   1:  PR[GP1:91,2] = PR[GP1:90,2] + -26.555;
   1:L PR[91] 10mm/sec CNT100;
   1:  PR[GP1:91,1] = PR[GP1:90,1] + 40.213;
   1:  PR[GP1:91,2] = PR[GP1:90,2] + -24.982;
   1:L PR[91] 10mm/sec CNT100;
   1:  PR[GP1:91,1] = PR[GP1:90,1] + 40.837;
   1:  PR[GP1:91,2] = PR[GP1:90,2] + -23.165;
   1:L PR[91] 10mm/sec CNT100;
   1:  PR[GP1:91,1] = PR[GP1:90,1] + 41.205;
   1:  PR[GP1:91,2] = PR[GP1:90,2] + -22.033;
   1:L PR[91] 10mm/sec CNT100;
   1:  PR[GP1:91,1] = PR[GP1:90,1] + 41.473;
   1:  PR[GP1:91,2] = PR[GP1:90,2] + -19.935;
   1:L PR[91] 10mm/sec CNT100;
   1:  PR[GP1:91,1] = PR[GP1:90,1] + 41.556;
   1:  PR[GP1:91,2] = PR[GP1:90,2] + -19.063;
   1:L PR[91] 10mm/sec CNT100;
   1:  PR[GP1:91,1] = PR[GP1:90,1] + 41.398;
   1:  PR[GP1:91,2] = PR[GP1:90,2] + -16.553;
   1:L PR[91] 10mm/sec CNT100;
   1:  PR[GP1:91,1] = PR[GP1:90,1] + 41.349;
   1:  PR[GP1:91,2] = PR[GP1:90,2] + -15.980;
   1:L PR[91] 10mm/sec CNT100;
   1:  PR[GP1:91,1] = PR[GP1:90,1] + 40.579;
   1:  PR[GP1:91,2] = PR[GP1:90,2] + -12.781;
   1:L PR[91] 10mm/sec CNT100;
   1:  PR[GP1:91,1] = PR[GP1:90,1] + 40.451;
   1:  PR[GP1:91,2] = PR[GP1:90,2] + -12.456;
   1:L PR[91] 10mm/sec CNT100;
   1:  PR[GP1:91,1] = PR[GP1:90,1] + 39.480;
   1:  PR[GP1:91,2] = PR[GP1:90,2] + -10.268;
   1:L PR[91] 10mm/sec CNT100;
   1:  PR[GP1:91,1] = PR[GP1:90,1] + 39.401;
   1:  PR[GP1:91,2] = PR[GP1:90,2] + -10.113;
   1:L PR[91] 10mm/sec CNT100;
   1:  PR[GP1:91,1] = PR[GP1:90,1] + 37.962;
   1:  PR[GP1:91,2] = PR[GP1:90,2] + -7.702;
   1:L PR[91] 10mm/sec CNT100;
   1:  PR[GP1:91,1] = PR[GP1:90,1] + 37.582;
   1:  PR[GP1:91,2] = PR[GP1:90,2] + -7.166;
   1:L PR[91] 10mm/sec CNT100;
   1:  PR[GP1:91,1] = PR[GP1:90,1] + 36.402;
   1:  PR[GP1:91,2] = PR[GP1:90,2] + -5.604;
   1:L PR[91] 10mm/sec CNT100;
   1:  PR[GP1:91,1] = PR[GP1:90,1] + 35.683;
   1:  PR[GP1:91,2] = PR[GP1:90,2] + -4.745;
   1:L PR[91] 10mm/sec CNT100;
   1:  PR[GP1:91,1] = PR[GP1:90,1] + 34.717;
   1:  PR[GP1:91,2] = PR[GP1:90,2] + -3.709;
   1:L PR[91] 10mm/sec CNT100;
   1:  PR[GP1:91,1] = PR[GP1:90,1] + 33.533;
   1:  PR[GP1:91,2] = PR[GP1:90,2] + -2.515;
   1:L PR[91] 10mm/sec CNT100;
   1:  PR[GP1:91,1] = PR[GP1:90,1] + 32.203;
   1:  PR[GP1:91,2] = PR[GP1:90,2] + -1.332;
   1:L PR[91] 10mm/sec CNT100;
   1:  PR[GP1:91,1] = PR[GP1:90,1] + 29.155;
   1:  PR[GP1:91,2] = PR[GP1:90,2] + 0.929;
   1:L PR[91] 10mm/sec CNT100;
   1:  PR[GP1:91,1] = PR[GP1:90,1] + 29.129;
   1:  PR[GP1:91,2] = PR[GP1:90,2] + 0.967;
   1:L PR[91] 10mm/sec CNT100;
   1:  PR[GP1:91,1] = PR[GP1:90,1] + 28.740;
   1:  PR[GP1:91,2] = PR[GP1:90,2] + 1.225;
   1:L PR[91] 10mm/sec CNT100;
   1:  PR[GP1:91,1] = PR[GP1:90,1] + 28.686;
   1:  PR[GP1:91,2] = PR[GP1:90,2] + 1.277;
   1:L PR[91] 10mm/sec CNT100;
   1:  PR[GP1:91,1] = PR[GP1:90,1] + 28.580;
   1:  PR[GP1:91,2] = PR[GP1:90,2] + 1.338;
   1:L PR[91] 10mm/sec CNT100;
   1:  PR[GP1:91,1] = PR[GP1:90,1] + 28.013;
   1:  PR[GP1:91,2] = PR[GP1:90,2] + 1.741;
   1:L PR[91] 10mm/sec CNT100;
   1:  PR[GP1:91,1] = PR[GP1:90,1] + 27.398;
   1:  PR[GP1:91,2] = PR[GP1:90,2] + 2.081;
   1:L PR[91] 10mm/sec CNT100;
   1:  PR[GP1:91,1] = PR[GP1:90,1] + 27.237;
   1:  PR[GP1:91,2] = PR[GP1:90,2] + 2.153;
   1:L PR[91] 10mm/sec CNT100;
   1:  PR[GP1:91,1] = PR[GP1:90,1] + 25.745;
   1:  PR[GP1:91,2] = PR[GP1:90,2] + 3.172;
   1:L PR[91] 10mm/sec CNT100;
   1:  PR[GP1:91,1] = PR[GP1:90,1] + 23.344;
   1:  PR[GP1:91,2] = PR[GP1:90,2] + 4.304;
   1:L PR[91] 10mm/sec CNT100;
   1:  PR[GP1:91,1] = PR[GP1:90,1] + 22.049;
   1:  PR[GP1:91,2] = PR[GP1:90,2] + 4.950;
   1:L PR[91] 10mm/sec CNT100;
   1:  PR[GP1:91,1] = PR[GP1:90,1] + 20.978;
   1:  PR[GP1:91,2] = PR[GP1:90,2] + 5.264;
   1:L PR[91] 10mm/sec CNT100;
   1:  PR[GP1:91,1] = PR[GP1:90,1] + 18.240;
   1:  PR[GP1:91,2] = PR[GP1:90,2] + 6.115;
   1:L PR[91] 10mm/sec CNT100;
   1:  PR[GP1:91,1] = PR[GP1:90,1] + 14.410;
   1:  PR[GP1:91,2] = PR[GP1:90,2] + 6.611;
   1:L PR[91] 10mm/sec CNT100;
   1:  PR[GP1:91,1] = PR[GP1:90,1] + 12.441;
   1:  PR[GP1:91,2] = PR[GP1:90,2] + 6.605;
   1:L PR[91] 10mm/sec CNT100;
   1:  PR[GP1:91,1] = PR[GP1:90,1] + 8.605;
   1:  PR[GP1:91,2] = PR[GP1:90,2] + 6.454;
   1:L PR[91] 10mm/sec CNT100;
   1:  PR[GP1:91,1] = PR[GP1:90,1] + 7.443;
   1:  PR[GP1:91,2] = PR[GP1:90,2] + 6.272;
   1:L PR[91] 10mm/sec CNT100;
   1:  PR[GP1:91,1] = PR[GP1:90,1] + 4.759;
   1:  PR[GP1:91,2] = PR[GP1:90,2] + 5.733;
   1:L PR[91] 10mm/sec CNT100;
   1:  PR[GP1:91,1] = PR[GP1:90,1] + 2.825;
   1:  PR[GP1:91,2] = PR[GP1:90,2] + 5.026;
   1:L PR[91] 10mm/sec CNT100;
   1:  PR[GP1:91,1] = PR[GP1:90,1] + 1.085;
   1:  PR[GP1:91,2] = PR[GP1:90,2] + 4.344;
   1:L PR[91] 10mm/sec CNT100;
   1:  PR[GP1:91,1] = PR[GP1:90,1] + 0.917;
   1:  PR[GP1:91,2] = PR[GP1:90,2] + 4.256;
   1:L PR[91] 10mm/sec CNT100;
   1:  PR[GP1:91,1] = PR[GP1:90,1] + -1.994;
   1:  PR[GP1:91,2] = PR[GP1:90,2] + 2.387;
   1:L PR[91] 10mm/sec CNT100;
   1:  PR[GP1:91,1] = PR[GP1:90,1] + -2.585;
   1:  PR[GP1:91,2] = PR[GP1:90,2] + 1.867;
   1:L PR[91] 10mm/sec CNT100;
   1:  PR[GP1:91,1] = PR[GP1:90,1] + -4.416;
   1:  PR[GP1:91,2] = PR[GP1:90,2] + -0.110;
   1:L PR[91] 10mm/sec CNT100;
   1:  PR[GP1:91,1] = PR[GP1:90,1] + -4.794;
   1:  PR[GP1:91,2] = PR[GP1:90,2] + -0.576;
   1:L PR[91] 10mm/sec CNT100;
   1:  PR[GP1:91,1] = PR[GP1:90,1] + -5.085;
   1:  PR[GP1:91,2] = PR[GP1:90,2] + -1.098;
   1:L PR[91] 10mm/sec CNT100;
   1:  PR[GP1:91,1] = PR[GP1:90,1] + -6.371;
   1:  PR[GP1:91,2] = PR[GP1:90,2] + -3.548;
   1:L PR[91] 10mm/sec CNT100;
   1:  PR[GP1:91,1] = PR[GP1:90,1] + -6.544;
   1:  PR[GP1:91,2] = PR[GP1:90,2] + -4.032;
   1:L PR[91] 10mm/sec CNT100;
   1:  PR[GP1:91,1] = PR[GP1:90,1] + -7.168;
   1:  PR[GP1:91,2] = PR[GP1:90,2] + -6.722;
   1:L PR[91] 10mm/sec CNT100;
   1:  PR[GP1:91,1] = PR[GP1:90,1] + -7.277;
   1:  PR[GP1:91,2] = PR[GP1:90,2] + -7.313;
   1:L PR[91] 10mm/sec CNT100;
   1:  PR[GP1:91,1] = PR[GP1:90,1] + -7.289;
   1:  PR[GP1:91,2] = PR[GP1:90,2] + -7.916;
   1:L PR[91] 10mm/sec CNT100;
   1:  PR[GP1:91,1] = PR[GP1:90,1] + -7.146;
   1:  PR[GP1:91,2] = PR[GP1:90,2] + -10.619;
   1:L PR[91] 10mm/sec CNT100;
   1:  PR[GP1:91,1] = PR[GP1:90,1] + -7.020;
   1:  PR[GP1:91,2] = PR[GP1:90,2] + -11.395;
   1:L PR[91] 10mm/sec CNT100;
   1:  PR[GP1:91,1] = PR[GP1:90,1] + -6.890;
   1:  PR[GP1:91,2] = PR[GP1:90,2] + -11.888;
   1:L PR[91] 10mm/sec CNT100;
   1:  PR[GP1:91,1] = PR[GP1:90,1] + -5.780;
   1:  PR[GP1:91,2] = PR[GP1:90,2] + -15.094;
   1:L PR[91] 10mm/sec CNT100;
   1:  PR[GP1:91,1] = PR[GP1:90,1] + -4.734;
   1:  PR[GP1:91,2] = PR[GP1:90,2] + -16.207;
   1:  PR[GP1:91,3] = PR[GP1:90,3] + 64.900;
   1:L PR[91] 10mm/sec CNT100;
   1:  PR[GP1:91,1] = PR[GP1:90,1] + -4.405;
   1:  PR[GP1:91,2] = PR[GP1:90,2] + -16.913;
   1:L PR[91] 10mm/sec CNT100;
   1:  PR[GP1:91,1] = PR[GP1:90,1] + -2.796;
   1:  PR[GP1:91,2] = PR[GP1:90,2] + -19.611;
   1:L PR[91] 10mm/sec CNT100;
   1:  PR[GP1:91,1] = PR[GP1:90,1] + -1.034;
   1:  PR[GP1:91,2] = PR[GP1:90,2] + -22.053;
   1:L PR[91] 10mm/sec CNT100;
   1:  PR[GP1:91,1] = PR[GP1:90,1] + 0.730;
   1:  PR[GP1:91,2] = PR[GP1:90,2] + -23.964;
   1:L PR[91] 10mm/sec CNT100;
   1:  PR[GP1:91,1] = PR[GP1:90,1] + 1.619;
   1:  PR[GP1:91,2] = PR[GP1:90,2] + -24.885;
   1:L PR[91] 10mm/sec CNT100;
   1:  PR[GP1:91,1] = PR[GP1:90,1] + 5.191;
   1:  PR[GP1:91,2] = PR[GP1:90,2] + -27.678;
   1:L PR[91] 10mm/sec CNT100;
   1:  PR[GP1:91,1] = PR[GP1:90,1] + 5.925;
   1:  PR[GP1:91,2] = PR[GP1:90,2] + -28.223;
   1:L PR[91] 10mm/sec CNT100;
   1:  PR[GP1:91,1] = PR[GP1:90,1] + 8.045;
   1:  PR[GP1:91,2] = PR[GP1:90,2] + -29.365;
   1:L PR[91] 10mm/sec CNT100;
   1:  PR[GP1:91,1] = PR[GP1:90,1] + 10.874;
   1:  PR[GP1:91,2] = PR[GP1:90,2] + -31.023;
   1:L PR[91] 10mm/sec CNT100;
   1:  PR[GP1:91,1] = PR[GP1:90,1] + 17.152;
   1:  PR[GP1:91,2] = PR[GP1:90,2] + -33.416;
   1:L PR[91] 10mm/sec CNT100;
   1:  PR[GP1:91,1] = PR[GP1:90,1] + 21.716;
   1:  PR[GP1:91,2] = PR[GP1:90,2] + -34.314;
   1:L PR[91] 10mm/sec CNT100;
   1:  PR[GP1:91,1] = PR[GP1:90,1] + 25.157;
   1:  PR[GP1:91,2] = PR[GP1:90,2] + -34.513;
   1:L PR[91] 10mm/sec CNT100;
   1:  PR[GP1:91,1] = PR[GP1:90,1] + 25.469;
   1:  PR[GP1:91,2] = PR[GP1:90,2] + -34.516;
   1:L PR[91] 10mm/sec CNT100;
   1:  PR[GP1:91,1] = PR[GP1:90,1] + 26.721;
   1:  PR[GP1:91,2] = PR[GP1:90,2] + -34.412;
   1:L PR[91] 10mm/sec CNT100;
   1:  PR[GP1:91,1] = PR[GP1:90,1] + 28.056;
   1:  PR[GP1:91,2] = PR[GP1:90,2] + -34.239;
   1:L PR[91] 10mm/sec CNT100;
   1:  PR[GP1:91,1] = PR[GP1:90,1] + 29.127;
   1:  PR[GP1:91,2] = PR[GP1:90,2] + -34.122;
   1:L PR[91] 10mm/sec CNT100;
   1:  PR[GP1:91,1] = PR[GP1:90,1] + 31.447;
   1:  PR[GP1:91,2] = PR[GP1:90,2] + -33.504;
   1:L PR[91] 10mm/sec CNT100;
   1:  PR[GP1:91,1] = PR[GP1:90,1] + 33.162;
   1:  PR[GP1:91,2] = PR[GP1:90,2] + -32.841;
   1:L PR[91] 10mm/sec CNT100;
   1:  PR[GP1:91,1] = PR[GP1:90,1] + 35.063;
   1:  PR[GP1:91,2] = PR[GP1:90,2] + -31.964;
   1:L PR[91] 10mm/sec CNT100;
   1:  PR[GP1:91,1] = PR[GP1:90,1] + 36.348;
   1:  PR[GP1:91,2] = PR[GP1:90,2] + -31.049;
   1:L PR[91] 10mm/sec CNT100;
   1:  PR[GP1:91,1] = PR[GP1:90,1] + 38.180;
   1:  PR[GP1:91,2] = PR[GP1:90,2] + -29.609;
   1:L PR[91] 10mm/sec CNT100;
   1:  PR[GP1:91,1] = PR[GP1:90,1] + 39.188;
   1:  PR[GP1:91,2] = PR[GP1:90,2] + -28.533;
   1:L PR[91] 10mm/sec CNT100;
   1:  PR[GP1:91,1] = PR[GP1:90,1] + 40.396;
   1:  PR[GP1:91,2] = PR[GP1:90,2] + -26.733;
   1:L PR[91] 10mm/sec CNT100;
   1:  PR[GP1:91,1] = PR[GP1:90,1] + 41.135;
   1:  PR[GP1:91,2] = PR[GP1:90,2] + -25.505;
   1:L PR[91] 10mm/sec CNT100;
   1:  PR[GP1:91,1] = PR[GP1:90,1] + 41.624;
   1:  PR[GP1:91,2] = PR[GP1:90,2] + -24.084;
   1:L PR[91] 10mm/sec CNT100;
   1:  PR[GP1:91,1] = PR[GP1:90,1] + 42.143;
   1:  PR[GP1:91,2] = PR[GP1:90,2] + -22.487;
   1:L PR[91] 10mm/sec CNT100;
   1:  PR[GP1:91,1] = PR[GP1:90,1] + 42.352;
   1:  PR[GP1:91,2] = PR[GP1:90,2] + -20.843;
   1:L PR[91] 10mm/sec CNT100;
   1:  PR[GP1:91,1] = PR[GP1:90,1] + 42.481;
   1:  PR[GP1:91,2] = PR[GP1:90,2] + -19.511;
   1:L PR[91] 10mm/sec CNT100;
   1:  PR[GP1:91,1] = PR[GP1:90,1] + 42.356;
   1:  PR[GP1:91,2] = PR[GP1:90,2] + -17.540;
   1:L PR[91] 10mm/sec CNT100;
   1:  PR[GP1:91,1] = PR[GP1:90,1] + 42.263;
   1:  PR[GP1:91,2] = PR[GP1:90,2] + -16.448;
   1:L PR[91] 10mm/sec CNT100;
   1:  PR[GP1:91,1] = PR[GP1:90,1] + 41.502;
   1:  PR[GP1:91,2] = PR[GP1:90,2] + -13.304;
   1:L PR[91] 10mm/sec CNT100;
   1:  PR[GP1:91,1] = PR[GP1:90,1] + 40.447;
   1:  PR[GP1:91,2] = PR[GP1:90,2] + -10.638;
   1:L PR[91] 10mm/sec CNT100;
   1:  PR[GP1:91,1] = PR[GP1:90,1] + 40.348;
   1:  PR[GP1:91,2] = PR[GP1:90,2] + -10.456;
   1:L PR[91] 10mm/sec CNT100;
   1:  PR[GP1:91,1] = PR[GP1:90,1] + 38.964;
   1:  PR[GP1:91,2] = PR[GP1:90,2] + -8.136;
   1:L PR[91] 10mm/sec CNT100;
   1:  PR[GP1:91,1] = PR[GP1:90,1] + 37.309;
   1:  PR[GP1:91,2] = PR[GP1:90,2] + -5.928;
   1:L PR[91] 10mm/sec CNT100;
   1:  PR[GP1:91,1] = PR[GP1:90,1] + 36.811;
   1:  PR[GP1:91,2] = PR[GP1:90,2] + -5.332;
   1:L PR[91] 10mm/sec CNT100;
   1:  PR[GP1:91,1] = PR[GP1:90,1] + 35.547;
   1:  PR[GP1:91,2] = PR[GP1:90,2] + -3.977;
   1:L PR[91] 10mm/sec CNT100;
   1:  PR[GP1:91,1] = PR[GP1:90,1] + 34.614;
   1:  PR[GP1:91,2] = PR[GP1:90,2] + -3.035;
   1:L PR[91] 10mm/sec CNT100;
   1:  PR[GP1:91,1] = PR[GP1:90,1] + 34.115;
   1:  PR[GP1:91,2] = PR[GP1:90,2] + -2.587;
   1:L PR[91] 10mm/sec CNT100;
   1:  PR[GP1:91,1] = PR[GP1:90,1] + 33.026;
   1:  PR[GP1:91,2] = PR[GP1:90,2] + -1.629;
   1:L PR[91] 10mm/sec CNT100;
   1:  PR[GP1:91,1] = PR[GP1:90,1] + 29.616;
   1:  PR[GP1:91,2] = PR[GP1:90,2] + 0.891;
   1:L PR[91] 10mm/sec CNT100;
   1:  PR[GP1:91,1] = PR[GP1:90,1] + 29.210;
   1:  PR[GP1:91,2] = PR[GP1:90,2] + 1.129;
   1:L PR[91] 10mm/sec CNT100;
   1:  PR[GP1:91,1] = PR[GP1:90,1] + 28.380;
   1:  PR[GP1:91,2] = PR[GP1:90,2] + 1.577;
   1:L PR[91] 10mm/sec CNT100;
   1:  PR[GP1:91,1] = PR[GP1:90,1] + 27.313;
   1:  PR[GP1:91,2] = PR[GP1:90,2] + 2.246;
   1:L PR[91] 10mm/sec CNT100;
   1:  PR[GP1:91,1] = PR[GP1:90,1] + 27.035;
   1:  PR[GP1:91,2] = PR[GP1:90,2] + 2.400;
   1:L PR[91] 10mm/sec CNT100;
   1:  PR[GP1:91,1] = PR[GP1:90,1] + 26.810;
   1:  PR[GP1:91,2] = PR[GP1:90,2] + 2.500;
   1:L PR[91] 10mm/sec CNT100;
   1:  PR[GP1:91,1] = PR[GP1:90,1] + 26.285;
   1:  PR[GP1:91,2] = PR[GP1:90,2] + 2.859;
   1:L PR[91] 10mm/sec CNT100;
   1:  PR[GP1:91,1] = PR[GP1:90,1] + 25.433;
   1:  PR[GP1:91,2] = PR[GP1:90,2] + 3.280;
   1:L PR[91] 10mm/sec CNT100;
   1:  PR[GP1:91,1] = PR[GP1:90,1] + 24.915;
   1:  PR[GP1:91,2] = PR[GP1:90,2] + 3.465;
   1:L PR[91] 10mm/sec CNT100;
   1:  PR[GP1:91,1] = PR[GP1:90,1] + 22.555;
   1:  PR[GP1:91,2] = PR[GP1:90,2] + 4.596;
   1:L PR[91] 10mm/sec CNT100;
   1:  PR[GP1:91,1] = PR[GP1:90,1] + 20.074;
   1:  PR[GP1:91,2] = PR[GP1:90,2] + 5.324;
   1:L PR[91] 10mm/sec CNT100;
   1:  PR[GP1:91,1] = PR[GP1:90,1] + 18.724;
   1:  PR[GP1:91,2] = PR[GP1:90,2] + 5.743;
   1:L PR[91] 10mm/sec CNT100;
   1:  PR[GP1:91,1] = PR[GP1:90,1] + 17.211;
   1:  PR[GP1:91,2] = PR[GP1:90,2] + 5.924;
   1:L PR[91] 10mm/sec CNT100;
   1:  PR[GP1:91,1] = PR[GP1:90,1] + 14.871;
   1:  PR[GP1:91,2] = PR[GP1:90,2] + 6.230;
   1:L PR[91] 10mm/sec CNT100;
   1:  PR[GP1:91,1] = PR[GP1:90,1] + 13.046;
   1:  PR[GP1:91,2] = PR[GP1:90,2] + 6.243;
   1:L PR[91] 10mm/sec CNT100;
   1:  PR[GP1:91,1] = PR[GP1:90,1] + 9.327;
   1:  PR[GP1:91,2] = PR[GP1:90,2] + 6.100;
   1:L PR[91] 10mm/sec CNT100;
   1:  PR[GP1:91,1] = PR[GP1:90,1] + 8.773;
   1:  PR[GP1:91,2] = PR[GP1:90,2] + 6.013;
   1:L PR[91] 10mm/sec CNT100;
   1:  PR[GP1:91,1] = PR[GP1:90,1] + 5.547;
   1:  PR[GP1:91,2] = PR[GP1:90,2] + 5.366;
   1:L PR[91] 10mm/sec CNT100;
   1:  PR[GP1:91,1] = PR[GP1:90,1] + 4.176;
   1:  PR[GP1:91,2] = PR[GP1:90,2] + 4.864;
   1:L PR[91] 10mm/sec CNT100;
   1:  PR[GP1:91,1] = PR[GP1:90,1] + 1.935;
   1:  PR[GP1:91,2] = PR[GP1:90,2] + 3.985;
   1:L PR[91] 10mm/sec CNT100;
   1:  PR[GP1:91,1] = PR[GP1:90,1] + 1.703;
   1:  PR[GP1:91,2] = PR[GP1:90,2] + 3.865;
   1:L PR[91] 10mm/sec CNT100;
   1:  PR[GP1:91,1] = PR[GP1:90,1] + -1.041;
   1:  PR[GP1:91,2] = PR[GP1:90,2] + 2.105;
   1:L PR[91] 10mm/sec CNT100;
   1:  PR[GP1:91,1] = PR[GP1:90,1] + -1.902;
   1:  PR[GP1:91,2] = PR[GP1:90,2] + 1.348;
   1:L PR[91] 10mm/sec CNT100;
   1:  PR[GP1:91,1] = PR[GP1:90,1] + -3.341;
   1:  PR[GP1:91,2] = PR[GP1:90,2] + -0.206;
   1:L PR[91] 10mm/sec CNT100;
   1:  PR[GP1:91,1] = PR[GP1:90,1] + -3.962;
   1:  PR[GP1:91,2] = PR[GP1:90,2] + -0.973;
   1:L PR[91] 10mm/sec CNT100;
   1:  PR[GP1:91,1] = PR[GP1:90,1] + -4.439;
   1:  PR[GP1:91,2] = PR[GP1:90,2] + -1.824;
   1:L PR[91] 10mm/sec CNT100;
   1:  PR[GP1:91,1] = PR[GP1:90,1] + -5.449;
   1:  PR[GP1:91,2] = PR[GP1:90,2] + -3.751;
   1:L PR[91] 10mm/sec CNT100;
   1:  PR[GP1:91,1] = PR[GP1:90,1] + -5.752;
   1:  PR[GP1:91,2] = PR[GP1:90,2] + -4.595;
   1:L PR[91] 10mm/sec CNT100;
   1:  PR[GP1:91,1] = PR[GP1:90,1] + -6.243;
   1:  PR[GP1:91,2] = PR[GP1:90,2] + -6.711;
   1:L PR[91] 10mm/sec CNT100;
   1:  PR[GP1:91,1] = PR[GP1:90,1] + -6.418;
   1:  PR[GP1:91,2] = PR[GP1:90,2] + -7.664;
   1:L PR[91] 10mm/sec CNT100;
   1:  PR[GP1:91,1] = PR[GP1:90,1] + -6.437;
   1:  PR[GP1:91,2] = PR[GP1:90,2] + -8.641;
   1:L PR[91] 10mm/sec CNT100;
   1:  PR[GP1:91,1] = PR[GP1:90,1] + -6.325;
   1:  PR[GP1:91,2] = PR[GP1:90,2] + -10.765;
   1:L PR[91] 10mm/sec CNT100;
   1:  PR[GP1:91,1] = PR[GP1:90,1] + -6.147;
   1:  PR[GP1:91,2] = PR[GP1:90,2] + -11.863;
   1:L PR[91] 10mm/sec CNT100;
   1:  PR[GP1:91,1] = PR[GP1:90,1] + -6.138;
   1:  PR[GP1:91,2] = PR[GP1:90,2] + -11.898;
   1:L PR[91] 10mm/sec CNT100;
   1:  PR[GP1:91,1] = PR[GP1:90,1] + -4.973;
   1:  PR[GP1:91,2] = PR[GP1:90,2] + -15.416;
   1:L PR[91] 10mm/sec CNT100;
   1:  PR[GP1:91,1] = PR[GP1:90,1] + -3.994;
   1:  PR[GP1:91,2] = PR[GP1:90,2] + -16.372;
   1:  PR[GP1:91,3] = PR[GP1:90,3] + 66.000;
   1:L PR[91] 10mm/sec CNT100;
   1:  PR[GP1:91,1] = PR[GP1:90,1] + -3.394;
   1:  PR[GP1:91,2] = PR[GP1:90,2] + -17.660;
   1:L PR[91] 10mm/sec CNT100;
   1:  PR[GP1:91,1] = PR[GP1:90,1] + -2.220;
   1:  PR[GP1:91,2] = PR[GP1:90,2] + -19.628;
   1:L PR[91] 10mm/sec CNT100;
   1:  PR[GP1:91,1] = PR[GP1:90,1] + 0.080;
   1:  PR[GP1:91,2] = PR[GP1:90,2] + -22.816;
   1:L PR[91] 10mm/sec CNT100;
   1:  PR[GP1:91,1] = PR[GP1:90,1] + 1.368;
   1:  PR[GP1:91,2] = PR[GP1:90,2] + -24.212;
   1:L PR[91] 10mm/sec CNT100;
   1:  PR[GP1:91,1] = PR[GP1:90,1] + 2.418;
   1:  PR[GP1:91,2] = PR[GP1:90,2] + -25.298;
   1:L PR[91] 10mm/sec CNT100;
   1:  PR[GP1:91,1] = PR[GP1:90,1] + 6.705;
   1:  PR[GP1:91,2] = PR[GP1:90,2] + -28.646;
   1:L PR[91] 10mm/sec CNT100;
   1:  PR[GP1:91,1] = PR[GP1:90,1] + 7.013;
   1:  PR[GP1:91,2] = PR[GP1:90,2] + -28.812;
   1:L PR[91] 10mm/sec CNT100;
   1:  PR[GP1:91,1] = PR[GP1:90,1] + 11.732;
   1:  PR[GP1:91,2] = PR[GP1:90,2] + -31.577;
   1:L PR[91] 10mm/sec CNT100;
   1:  PR[GP1:91,1] = PR[GP1:90,1] + 18.232;
   1:  PR[GP1:91,2] = PR[GP1:90,2] + -34.059;
   1:L PR[91] 10mm/sec CNT100;
   1:  PR[GP1:91,1] = PR[GP1:90,1] + 22.586;
   1:  PR[GP1:91,2] = PR[GP1:90,2] + -34.911;
   1:L PR[91] 10mm/sec CNT100;
   1:  PR[GP1:91,1] = PR[GP1:90,1] + 25.143;
   1:  PR[GP1:91,2] = PR[GP1:90,2] + -35.058;
   1:L PR[91] 10mm/sec CNT100;
   1:  PR[GP1:91,1] = PR[GP1:90,1] + 26.073;
   1:  PR[GP1:91,2] = PR[GP1:90,2] + -35.091;
   1:L PR[91] 10mm/sec CNT100;
   1:  PR[GP1:91,1] = PR[GP1:90,1] + 27.886;
   1:  PR[GP1:91,2] = PR[GP1:90,2] + -34.856;
   1:L PR[91] 10mm/sec CNT100;
   1:  PR[GP1:91,1] = PR[GP1:90,1] + 30.291;
   1:  PR[GP1:91,2] = PR[GP1:90,2] + -34.593;
   1:L PR[91] 10mm/sec CNT100;
   1:  PR[GP1:91,1] = PR[GP1:90,1] + 31.974;
   1:  PR[GP1:91,2] = PR[GP1:90,2] + -34.145;
   1:L PR[91] 10mm/sec CNT100;
   1:  PR[GP1:91,1] = PR[GP1:90,1] + 34.587;
   1:  PR[GP1:91,2] = PR[GP1:90,2] + -33.135;
   1:L PR[91] 10mm/sec CNT100;
   1:  PR[GP1:91,1] = PR[GP1:90,1] + 35.964;
   1:  PR[GP1:91,2] = PR[GP1:90,2] + -32.500;
   1:L PR[91] 10mm/sec CNT100;
   1:  PR[GP1:91,1] = PR[GP1:90,1] + 36.892;
   1:  PR[GP1:91,2] = PR[GP1:90,2] + -31.839;
   1:L PR[91] 10mm/sec CNT100;
   1:  PR[GP1:91,1] = PR[GP1:90,1] + 39.268;
   1:  PR[GP1:91,2] = PR[GP1:90,2] + -29.972;
   1:L PR[91] 10mm/sec CNT100;
   1:  PR[GP1:91,1] = PR[GP1:90,1] + 39.990;
   1:  PR[GP1:91,2] = PR[GP1:90,2] + -29.202;
   1:L PR[91] 10mm/sec CNT100;
   1:  PR[GP1:91,1] = PR[GP1:90,1] + 41.526;
   1:  PR[GP1:91,2] = PR[GP1:90,2] + -26.912;
   1:L PR[91] 10mm/sec CNT100;
   1:  PR[GP1:91,1] = PR[GP1:90,1] + 42.058;
   1:  PR[GP1:91,2] = PR[GP1:90,2] + -26.028;
   1:L PR[91] 10mm/sec CNT100;
   1:  PR[GP1:91,1] = PR[GP1:90,1] + 42.410;
   1:  PR[GP1:91,2] = PR[GP1:90,2] + -25.003;
   1:L PR[91] 10mm/sec CNT100;
   1:  PR[GP1:91,1] = PR[GP1:90,1] + 43.081;
   1:  PR[GP1:91,2] = PR[GP1:90,2] + -22.941;
   1:L PR[91] 10mm/sec CNT100;
   1:  PR[GP1:91,1] = PR[GP1:90,1] + 43.232;
   1:  PR[GP1:91,2] = PR[GP1:90,2] + -21.752;
   1:L PR[91] 10mm/sec CNT100;
   1:  PR[GP1:91,1] = PR[GP1:90,1] + 43.405;
   1:  PR[GP1:91,2] = PR[GP1:90,2] + -19.959;
   1:L PR[91] 10mm/sec CNT100;
   1:  PR[GP1:91,1] = PR[GP1:90,1] + 43.314;
   1:  PR[GP1:91,2] = PR[GP1:90,2] + -18.526;
   1:L PR[91] 10mm/sec CNT100;
   1:  PR[GP1:91,1] = PR[GP1:90,1] + 43.177;
   1:  PR[GP1:91,2] = PR[GP1:90,2] + -16.916;
   1:L PR[91] 10mm/sec CNT100;
   1:  PR[GP1:91,1] = PR[GP1:90,1] + 42.426;
   1:  PR[GP1:91,2] = PR[GP1:90,2] + -13.828;
   1:L PR[91] 10mm/sec CNT100;
   1:  PR[GP1:91,1] = PR[GP1:90,1] + 41.351;
   1:  PR[GP1:91,2] = PR[GP1:90,2] + -11.122;
   1:L PR[91] 10mm/sec CNT100;
   1:  PR[GP1:91,1] = PR[GP1:90,1] + 40.038;
   1:  PR[GP1:91,2] = PR[GP1:90,2] + -8.690;
   1:L PR[91] 10mm/sec CNT100;
   1:  PR[GP1:91,1] = PR[GP1:90,1] + 39.962;
   1:  PR[GP1:91,2] = PR[GP1:90,2] + -8.563;
   1:L PR[91] 10mm/sec CNT100;
   1:  PR[GP1:91,1] = PR[GP1:90,1] + 38.218;
   1:  PR[GP1:91,2] = PR[GP1:90,2] + -6.253;
   1:L PR[91] 10mm/sec CNT100;
   1:  PR[GP1:91,1] = PR[GP1:90,1] + 37.938;
   1:  PR[GP1:91,2] = PR[GP1:90,2] + -5.919;
   1:L PR[91] 10mm/sec CNT100;
   1:  PR[GP1:91,1] = PR[GP1:90,1] + 36.376;
   1:  PR[GP1:91,2] = PR[GP1:90,2] + -4.244;
   1:L PR[91] 10mm/sec CNT100;
   1:  PR[GP1:91,1] = PR[GP1:90,1] + 35.698;
   1:  PR[GP1:91,2] = PR[GP1:90,2] + -3.559;
   1:L PR[91] 10mm/sec CNT100;
   1:  PR[GP1:91,1] = PR[GP1:90,1] + 33.847;
   1:  PR[GP1:91,2] = PR[GP1:90,2] + -1.925;
   1:L PR[91] 10mm/sec CNT100;
   1:  PR[GP1:91,1] = PR[GP1:90,1] + 31.640;
   1:  PR[GP1:91,2] = PR[GP1:90,2] + -0.287;
   1:L PR[91] 10mm/sec CNT100;
   1:  PR[GP1:91,1] = PR[GP1:90,1] + 30.597;
   1:  PR[GP1:91,2] = PR[GP1:90,2] + 0.463;
   1:L PR[91] 10mm/sec CNT100;
   1:  PR[GP1:91,1] = PR[GP1:90,1] + 29.500;
   1:  PR[GP1:91,2] = PR[GP1:90,2] + 1.104;
   1:L PR[91] 10mm/sec CNT100;
   1:  PR[GP1:91,1] = PR[GP1:90,1] + 27.410;
   1:  PR[GP1:91,2] = PR[GP1:90,2] + 2.233;
   1:L PR[91] 10mm/sec CNT100;
   1:  PR[GP1:91,1] = PR[GP1:90,1] + 26.928;
   1:  PR[GP1:91,2] = PR[GP1:90,2] + 2.534;
   1:L PR[91] 10mm/sec CNT100;
   1:  PR[GP1:91,1] = PR[GP1:90,1] + 26.078;
   1:  PR[GP1:91,2] = PR[GP1:90,2] + 2.912;
   1:L PR[91] 10mm/sec CNT100;
   1:  PR[GP1:91,1] = PR[GP1:90,1] + 25.264;
   1:  PR[GP1:91,2] = PR[GP1:90,2] + 3.316;
   1:L PR[91] 10mm/sec CNT100;
   1:  PR[GP1:91,1] = PR[GP1:90,1] + 24.344;
   1:  PR[GP1:91,2] = PR[GP1:90,2] + 3.645;
   1:L PR[91] 10mm/sec CNT100;
   1:  PR[GP1:91,1] = PR[GP1:90,1] + 23.068;
   1:  PR[GP1:91,2] = PR[GP1:90,2] + 4.254;
   1:L PR[91] 10mm/sec CNT100;
   1:  PR[GP1:91,1] = PR[GP1:90,1] + 22.587;
   1:  PR[GP1:91,2] = PR[GP1:90,2] + 4.408;
   1:L PR[91] 10mm/sec CNT100;
   1:  PR[GP1:91,1] = PR[GP1:90,1] + 22.054;
   1:  PR[GP1:91,2] = PR[GP1:90,2] + 4.526;
   1:L PR[91] 10mm/sec CNT100;
   1:  PR[GP1:91,1] = PR[GP1:90,1] + 19.208;
   1:  PR[GP1:91,2] = PR[GP1:90,2] + 5.372;
   1:L PR[91] 10mm/sec CNT100;
   1:  PR[GP1:91,1] = PR[GP1:90,1] + 15.337;
   1:  PR[GP1:91,2] = PR[GP1:90,2] + 5.847;
   1:L PR[91] 10mm/sec CNT100;
   1:  PR[GP1:91,1] = PR[GP1:90,1] + 13.575;
   1:  PR[GP1:91,2] = PR[GP1:90,2] + 5.880;
   1:L PR[91] 10mm/sec CNT100;
   1:  PR[GP1:91,1] = PR[GP1:90,1] + 10.065;
   1:  PR[GP1:91,2] = PR[GP1:90,2] + 5.746;
   1:L PR[91] 10mm/sec CNT100;
   1:  PR[GP1:91,1] = PR[GP1:90,1] + 6.335;
   1:  PR[GP1:91,2] = PR[GP1:90,2] + 4.998;
   1:L PR[91] 10mm/sec CNT100;
   1:  PR[GP1:91,1] = PR[GP1:90,1] + 5.527;
   1:  PR[GP1:91,2] = PR[GP1:90,2] + 4.703;
   1:L PR[91] 10mm/sec CNT100;
   1:  PR[GP1:91,1] = PR[GP1:90,1] + 2.784;
   1:  PR[GP1:91,2] = PR[GP1:90,2] + 3.627;
   1:L PR[91] 10mm/sec CNT100;
   1:  PR[GP1:91,1] = PR[GP1:90,1] + 2.489;
   1:  PR[GP1:91,2] = PR[GP1:90,2] + 3.473;
   1:L PR[91] 10mm/sec CNT100;
   1:  PR[GP1:91,1] = PR[GP1:90,1] + -0.089;
   1:  PR[GP1:91,2] = PR[GP1:90,2] + 1.822;
   1:L PR[91] 10mm/sec CNT100;
   1:  PR[GP1:91,1] = PR[GP1:90,1] + -1.218;
   1:  PR[GP1:91,2] = PR[GP1:90,2] + 0.829;
   1:L PR[91] 10mm/sec CNT100;
   1:  PR[GP1:91,1] = PR[GP1:90,1] + -2.266;
   1:  PR[GP1:91,2] = PR[GP1:90,2] + -0.303;
   1:L PR[91] 10mm/sec CNT100;
   1:  PR[GP1:91,1] = PR[GP1:90,1] + -3.131;
   1:  PR[GP1:91,2] = PR[GP1:90,2] + -1.370;
   1:L PR[91] 10mm/sec CNT100;
   1:  PR[GP1:91,1] = PR[GP1:90,1] + -3.792;
   1:  PR[GP1:91,2] = PR[GP1:90,2] + -2.551;
   1:L PR[91] 10mm/sec CNT100;
   1:  PR[GP1:91,1] = PR[GP1:90,1] + -4.528;
   1:  PR[GP1:91,2] = PR[GP1:90,2] + -3.954;
   1:L PR[91] 10mm/sec CNT100;
   1:  PR[GP1:91,1] = PR[GP1:90,1] + -4.960;
   1:  PR[GP1:91,2] = PR[GP1:90,2] + -5.159;
   1:L PR[91] 10mm/sec CNT100;
   1:  PR[GP1:91,1] = PR[GP1:90,1] + -5.318;
   1:  PR[GP1:91,2] = PR[GP1:90,2] + -6.701;
   1:L PR[91] 10mm/sec CNT100;
   1:  PR[GP1:91,1] = PR[GP1:90,1] + -5.559;
   1:  PR[GP1:91,2] = PR[GP1:90,2] + -8.014;
   1:L PR[91] 10mm/sec CNT100;
   1:  PR[GP1:91,1] = PR[GP1:90,1] + -5.585;
   1:  PR[GP1:91,2] = PR[GP1:90,2] + -9.366;
   1:L PR[91] 10mm/sec CNT100;
   1:  PR[GP1:91,1] = PR[GP1:90,1] + -5.504;
   1:  PR[GP1:91,2] = PR[GP1:90,2] + -10.911;
   1:L PR[91] 10mm/sec CNT100;
   1:  PR[GP1:91,1] = PR[GP1:90,1] + -5.355;
   1:  PR[GP1:91,2] = PR[GP1:90,2] + -11.828;
   1:L PR[91] 10mm/sec CNT100;
   1:  PR[GP1:91,1] = PR[GP1:90,1] + -5.280;
   1:  PR[GP1:91,2] = PR[GP1:90,2] + -12.349;
   1:L PR[91] 10mm/sec CNT100;
   1:  PR[GP1:91,1] = PR[GP1:90,1] + -4.420;
   1:  PR[GP1:91,2] = PR[GP1:90,2] + -14.964;
   1:L PR[91] 10mm/sec CNT100;
   1:  PR[GP1:91,1] = PR[GP1:90,1] + -3.255;
   1:  PR[GP1:91,2] = PR[GP1:90,2] + -16.536;
   1:  PR[GP1:91,3] = PR[GP1:90,3] + 67.100;
   1:L PR[91] 10mm/sec CNT100;
   1:  PR[GP1:91,1] = PR[GP1:90,1] + -2.383;
   1:  PR[GP1:91,2] = PR[GP1:90,2] + -18.407;
   1:L PR[91] 10mm/sec CNT100;
   1:  PR[GP1:91,1] = PR[GP1:90,1] + -1.645;
   1:  PR[GP1:91,2] = PR[GP1:90,2] + -19.646;
   1:L PR[91] 10mm/sec CNT100;
   1:  PR[GP1:91,1] = PR[GP1:90,1] + 1.194;
   1:  PR[GP1:91,2] = PR[GP1:90,2] + -23.579;
   1:L PR[91] 10mm/sec CNT100;
   1:  PR[GP1:91,1] = PR[GP1:90,1] + 2.006;
   1:  PR[GP1:91,2] = PR[GP1:90,2] + -24.459;
   1:L PR[91] 10mm/sec CNT100;
   1:  PR[GP1:91,1] = PR[GP1:90,1] + 3.217;
   1:  PR[GP1:91,2] = PR[GP1:90,2] + -25.712;
   1:L PR[91] 10mm/sec CNT100;
   1:  PR[GP1:91,1] = PR[GP1:90,1] + 6.189;
   1:  PR[GP1:91,2] = PR[GP1:90,2] + -28.036;
   1:L PR[91] 10mm/sec CNT100;
   1:  PR[GP1:91,1] = PR[GP1:90,1] + 7.234;
   1:  PR[GP1:91,2] = PR[GP1:90,2] + -28.930;
   1:L PR[91] 10mm/sec CNT100;
   1:  PR[GP1:91,1] = PR[GP1:90,1] + 9.127;
   1:  PR[GP1:91,2] = PR[GP1:90,2] + -30.102;
   1:L PR[91] 10mm/sec CNT100;
   1:  PR[GP1:91,1] = PR[GP1:90,1] + 12.590;
   1:  PR[GP1:91,2] = PR[GP1:90,2] + -32.130;
   1:L PR[91] 10mm/sec CNT100;
   1:  PR[GP1:91,1] = PR[GP1:90,1] + 19.312;
   1:  PR[GP1:91,2] = PR[GP1:90,2] + -34.703;
   1:L PR[91] 10mm/sec CNT100;
   1:  PR[GP1:91,1] = PR[GP1:90,1] + 23.450;
   1:  PR[GP1:91,2] = PR[GP1:90,2] + -35.506;
   1:L PR[91] 10mm/sec CNT100;
   1:  PR[GP1:91,1] = PR[GP1:90,1] + 26.575;
   1:  PR[GP1:91,2] = PR[GP1:90,2] + -35.621;
   1:L PR[91] 10mm/sec CNT100;
   1:  PR[GP1:91,1] = PR[GP1:90,1] + 27.716;
   1:  PR[GP1:91,2] = PR[GP1:90,2] + -35.473;
   1:L PR[91] 10mm/sec CNT100;
   1:  PR[GP1:91,1] = PR[GP1:90,1] + 31.454;
   1:  PR[GP1:91,2] = PR[GP1:90,2] + -35.065;
   1:L PR[91] 10mm/sec CNT100;
   1:  PR[GP1:91,1] = PR[GP1:90,1] + 32.501;
   1:  PR[GP1:91,2] = PR[GP1:90,2] + -34.786;
   1:L PR[91] 10mm/sec CNT100;
   1:  PR[GP1:91,1] = PR[GP1:90,1] + 36.012;
   1:  PR[GP1:91,2] = PR[GP1:90,2] + -33.429;
   1:L PR[91] 10mm/sec CNT100;
   1:  PR[GP1:91,1] = PR[GP1:90,1] + 36.865;
   1:  PR[GP1:91,2] = PR[GP1:90,2] + -33.035;
   1:L PR[91] 10mm/sec CNT100;
   1:  PR[GP1:91,1] = PR[GP1:90,1] + 37.435;
   1:  PR[GP1:91,2] = PR[GP1:90,2] + -32.629;
   1:L PR[91] 10mm/sec CNT100;
   1:  PR[GP1:91,1] = PR[GP1:90,1] + 40.356;
   1:  PR[GP1:91,2] = PR[GP1:90,2] + -30.335;
   1:L PR[91] 10mm/sec CNT100;
   1:  PR[GP1:91,1] = PR[GP1:90,1] + 40.792;
   1:  PR[GP1:91,2] = PR[GP1:90,2] + -29.870;
   1:L PR[91] 10mm/sec CNT100;
   1:  PR[GP1:91,1] = PR[GP1:90,1] + 42.656;
   1:  PR[GP1:91,2] = PR[GP1:90,2] + -27.090;
   1:L PR[91] 10mm/sec CNT100;
   1:  PR[GP1:91,1] = PR[GP1:90,1] + 42.978;
   1:  PR[GP1:91,2] = PR[GP1:90,2] + -26.555;
   1:L PR[91] 10mm/sec CNT100;
   1:  PR[GP1:91,1] = PR[GP1:90,1] + 44.019;
   1:  PR[GP1:91,2] = PR[GP1:90,2] + -23.393;
   1:L PR[91] 10mm/sec CNT100;
   1:  PR[GP1:91,1] = PR[GP1:90,1] + 44.112;
   1:  PR[GP1:91,2] = PR[GP1:90,2] + -22.660;
   1:L PR[91] 10mm/sec CNT100;
   1:  PR[GP1:91,1] = PR[GP1:90,1] + 44.329;
   1:  PR[GP1:91,2] = PR[GP1:90,2] + -20.407;
   1:L PR[91] 10mm/sec CNT100;
   1:  PR[GP1:91,1] = PR[GP1:90,1] + 44.273;
   1:  PR[GP1:91,2] = PR[GP1:90,2] + -19.513;
   1:L PR[91] 10mm/sec CNT100;
   1:  PR[GP1:91,1] = PR[GP1:90,1] + 44.091;
   1:  PR[GP1:91,2] = PR[GP1:90,2] + -17.384;
   1:L PR[91] 10mm/sec CNT100;
   1:  PR[GP1:91,1] = PR[GP1:90,1] + 43.349;
   1:  PR[GP1:91,2] = PR[GP1:90,2] + -14.352;
   1:L PR[91] 10mm/sec CNT100;
   1:  PR[GP1:91,1] = PR[GP1:90,1] + 42.256;
   1:  PR[GP1:91,2] = PR[GP1:90,2] + -11.605;
   1:L PR[91] 10mm/sec CNT100;
   1:  PR[GP1:91,1] = PR[GP1:90,1] + 41.333;
   1:  PR[GP1:91,2] = PR[GP1:90,2] + -9.896;
   1:L PR[91] 10mm/sec CNT100;
   1:  PR[GP1:91,1] = PR[GP1:90,1] + 40.837;
   1:  PR[GP1:91,2] = PR[GP1:90,2] + -8.992;
   1:L PR[91] 10mm/sec CNT100;
   1:  PR[GP1:91,1] = PR[GP1:90,1] + 39.625;
   1:  PR[GP1:91,2] = PR[GP1:90,2] + -7.238;
   1:L PR[91] 10mm/sec CNT100;
   1:  PR[GP1:91,1] = PR[GP1:90,1] + 39.056;
   1:  PR[GP1:91,2] = PR[GP1:90,2] + -6.496;
   1:L PR[91] 10mm/sec CNT100;
   1:  PR[GP1:91,1] = PR[GP1:90,1] + 37.205;
   1:  PR[GP1:91,2] = PR[GP1:90,2] + -4.511;
   1:L PR[91] 10mm/sec CNT100;
   1:  PR[GP1:91,1] = PR[GP1:90,1] + 36.780;
   1:  PR[GP1:91,2] = PR[GP1:90,2] + -4.082;
   1:L PR[91] 10mm/sec CNT100;
   1:  PR[GP1:91,1] = PR[GP1:90,1] + 34.669;
   1:  PR[GP1:91,2] = PR[GP1:90,2] + -2.221;
   1:L PR[91] 10mm/sec CNT100;
   1:  PR[GP1:91,1] = PR[GP1:90,1] + 33.268;
   1:  PR[GP1:91,2] = PR[GP1:90,2] + -1.181;
   1:L PR[91] 10mm/sec CNT100;
   1:  PR[GP1:91,1] = PR[GP1:90,1] + 31.575;
   1:  PR[GP1:91,2] = PR[GP1:90,2] + 0.038;
   1:L PR[91] 10mm/sec CNT100;
   1:  PR[GP1:91,1] = PR[GP1:90,1] + 29.790;
   1:  PR[GP1:91,2] = PR[GP1:90,2] + 1.079;
   1:L PR[91] 10mm/sec CNT100;
   1:  PR[GP1:91,1] = PR[GP1:90,1] + 27.575;
   1:  PR[GP1:91,2] = PR[GP1:90,2] + 2.276;
   1:L PR[91] 10mm/sec CNT100;
   1:  PR[GP1:91,1] = PR[GP1:90,1] + 27.005;
   1:  PR[GP1:91,2] = PR[GP1:90,2] + 2.540;
   1:L PR[91] 10mm/sec CNT100;
   1:  PR[GP1:91,1] = PR[GP1:90,1] + 26.472;
   1:  PR[GP1:91,2] = PR[GP1:90,2] + 2.731;
   1:L PR[91] 10mm/sec CNT100;
   1:  PR[GP1:91,1] = PR[GP1:90,1] + 24.273;
   1:  PR[GP1:91,2] = PR[GP1:90,2] + 3.639;
   1:L PR[91] 10mm/sec CNT100;
   1:  PR[GP1:91,1] = PR[GP1:90,1] + 23.770;
   1:  PR[GP1:91,2] = PR[GP1:90,2] + 3.826;
   1:L PR[91] 10mm/sec CNT100;
   1:  PR[GP1:91,1] = PR[GP1:90,1] + 23.594;
   1:  PR[GP1:91,2] = PR[GP1:90,2] + 3.910;
   1:L PR[91] 10mm/sec CNT100;
   1:  PR[GP1:91,1] = PR[GP1:90,1] + 22.396;
   1:  PR[GP1:91,2] = PR[GP1:90,2] + 4.295;
   1:L PR[91] 10mm/sec CNT100;
   1:  PR[GP1:91,1] = PR[GP1:90,1] + 21.586;
   1:  PR[GP1:91,2] = PR[GP1:90,2] + 4.486;
   1:L PR[91] 10mm/sec CNT100;
   1:  PR[GP1:91,1] = PR[GP1:90,1] + 21.181;
   1:  PR[GP1:91,2] = PR[GP1:90,2] + 4.563;
   1:L PR[91] 10mm/sec CNT100;
   1:  PR[GP1:91,1] = PR[GP1:90,1] + 19.662;
   1:  PR[GP1:91,2] = PR[GP1:90,2] + 5.014;
   1:L PR[91] 10mm/sec CNT100;
   1:  PR[GP1:91,1] = PR[GP1:90,1] + 18.744;
   1:  PR[GP1:91,2] = PR[GP1:90,2] + 5.154;
   1:L PR[91] 10mm/sec CNT100;
   1:  PR[GP1:91,1] = PR[GP1:90,1] + 16.109;
   1:  PR[GP1:91,2] = PR[GP1:90,2] + 5.443;
   1:L PR[91] 10mm/sec CNT100;
   1:  PR[GP1:91,1] = PR[GP1:90,1] + 14.539;
   1:  PR[GP1:91,2] = PR[GP1:90,2] + 5.511;
   1:L PR[91] 10mm/sec CNT100;
   1:  PR[GP1:91,1] = PR[GP1:90,1] + 14.110;
   1:  PR[GP1:91,2] = PR[GP1:90,2] + 5.516;
   1:L PR[91] 10mm/sec CNT100;
   1:  PR[GP1:91,1] = PR[GP1:90,1] + 11.845;
   1:  PR[GP1:91,2] = PR[GP1:90,2] + 5.430;
   1:L PR[91] 10mm/sec CNT100;
   1:  PR[GP1:91,1] = PR[GP1:90,1] + 10.838;
   1:  PR[GP1:91,2] = PR[GP1:90,2] + 5.366;
   1:L PR[91] 10mm/sec CNT100;
   1:  PR[GP1:91,1] = PR[GP1:90,1] + 7.122;
   1:  PR[GP1:91,2] = PR[GP1:90,2] + 4.630;
   1:L PR[91] 10mm/sec CNT100;
   1:  PR[GP1:91,1] = PR[GP1:90,1] + 6.877;
   1:  PR[GP1:91,2] = PR[GP1:90,2] + 4.541;
   1:L PR[91] 10mm/sec CNT100;
   1:  PR[GP1:91,1] = PR[GP1:90,1] + 3.634;
   1:  PR[GP1:91,2] = PR[GP1:90,2] + 3.268;
   1:L PR[91] 10mm/sec CNT100;
   1:  PR[GP1:91,1] = PR[GP1:90,1] + 3.274;
   1:  PR[GP1:91,2] = PR[GP1:90,2] + 3.081;
   1:L PR[91] 10mm/sec CNT100;
   1:  PR[GP1:91,1] = PR[GP1:90,1] + 0.864;
   1:  PR[GP1:91,2] = PR[GP1:90,2] + 1.540;
   1:L PR[91] 10mm/sec CNT100;
   1:  PR[GP1:91,1] = PR[GP1:90,1] + -0.535;
   1:  PR[GP1:91,2] = PR[GP1:90,2] + 0.310;
   1:L PR[91] 10mm/sec CNT100;
   1:  PR[GP1:91,1] = PR[GP1:90,1] + -1.191;
   1:  PR[GP1:91,2] = PR[GP1:90,2] + -0.399;
   1:L PR[91] 10mm/sec CNT100;
   1:  PR[GP1:91,1] = PR[GP1:90,1] + -2.299;
   1:  PR[GP1:91,2] = PR[GP1:90,2] + -1.766;
   1:L PR[91] 10mm/sec CNT100;
   1:  PR[GP1:91,1] = PR[GP1:90,1] + -3.145;
   1:  PR[GP1:91,2] = PR[GP1:90,2] + -3.277;
   1:L PR[91] 10mm/sec CNT100;
   1:  PR[GP1:91,1] = PR[GP1:90,1] + -3.606;
   1:  PR[GP1:91,2] = PR[GP1:90,2] + -4.157;
   1:L PR[91] 10mm/sec CNT100;
   1:  PR[GP1:91,1] = PR[GP1:90,1] + -4.168;
   1:  PR[GP1:91,2] = PR[GP1:90,2] + -5.723;
   1:L PR[91] 10mm/sec CNT100;
   1:  PR[GP1:91,1] = PR[GP1:90,1] + -4.392;
   1:  PR[GP1:91,2] = PR[GP1:90,2] + -6.690;
   1:L PR[91] 10mm/sec CNT100;
   1:  PR[GP1:91,1] = PR[GP1:90,1] + -4.700;
   1:  PR[GP1:91,2] = PR[GP1:90,2] + -8.365;
   1:L PR[91] 10mm/sec CNT100;
   1:  PR[GP1:91,1] = PR[GP1:90,1] + -4.734;
   1:  PR[GP1:91,2] = PR[GP1:90,2] + -10.091;
   1:L PR[91] 10mm/sec CNT100;
   1:  PR[GP1:91,1] = PR[GP1:90,1] + -4.683;
   1:  PR[GP1:91,2] = PR[GP1:90,2] + -11.057;
   1:L PR[91] 10mm/sec CNT100;
   1:  PR[GP1:91,1] = PR[GP1:90,1] + -4.590;
   1:  PR[GP1:91,2] = PR[GP1:90,2] + -11.633;
   1:L PR[91] 10mm/sec CNT100;
   1:  PR[GP1:91,1] = PR[GP1:90,1] + -4.412;
   1:  PR[GP1:91,2] = PR[GP1:90,2] + -12.855;
   1:L PR[91] 10mm/sec CNT100;
   1:  PR[GP1:91,1] = PR[GP1:90,1] + -3.868;
   1:  PR[GP1:91,2] = PR[GP1:90,2] + -14.510;
   1:L PR[91] 10mm/sec CNT100;
   1:  PR[GP1:91,1] = PR[GP1:90,1] + -2.515;
   1:  PR[GP1:91,2] = PR[GP1:90,2] + -16.701;
   1:  PR[GP1:91,3] = PR[GP1:90,3] + 68.200;
   1:L PR[91] 10mm/sec CNT100;
   1:  PR[GP1:91,1] = PR[GP1:90,1] + -1.373;
   1:  PR[GP1:91,2] = PR[GP1:90,2] + -19.154;
   1:L PR[91] 10mm/sec CNT100;
   1:  PR[GP1:91,1] = PR[GP1:90,1] + -1.069;
   1:  PR[GP1:91,2] = PR[GP1:90,2] + -19.664;
   1:L PR[91] 10mm/sec CNT100;
   1:  PR[GP1:91,1] = PR[GP1:90,1] + 2.304;
   1:  PR[GP1:91,2] = PR[GP1:90,2] + -24.337;
   1:L PR[91] 10mm/sec CNT100;
   1:  PR[GP1:91,1] = PR[GP1:90,1] + 4.017;
   1:  PR[GP1:91,2] = PR[GP1:90,2] + -26.127;
   1:L PR[91] 10mm/sec CNT100;
   1:  PR[GP1:91,1] = PR[GP1:90,1] + 5.297;
   1:  PR[GP1:91,2] = PR[GP1:90,2] + -27.128;
   1:L PR[91] 10mm/sec CNT100;
   1:  PR[GP1:91,1] = PR[GP1:90,1] + 7.670;
   1:  PR[GP1:91,2] = PR[GP1:90,2] + -29.157;
   1:L PR[91] 10mm/sec CNT100;
   1:  PR[GP1:91,1] = PR[GP1:90,1] + 11.968;
   1:  PR[GP1:91,2] = PR[GP1:90,2] + -31.818;
   1:L PR[91] 10mm/sec CNT100;
   1:  PR[GP1:91,1] = PR[GP1:90,1] + 13.448;
   1:  PR[GP1:91,2] = PR[GP1:90,2] + -32.684;
   1:L PR[91] 10mm/sec CNT100;
   1:  PR[GP1:91,1] = PR[GP1:90,1] + 20.392;
   1:  PR[GP1:91,2] = PR[GP1:90,2] + -35.346;
   1:L PR[91] 10mm/sec CNT100;
   1:  PR[GP1:91,1] = PR[GP1:90,1] + 22.229;
   1:  PR[GP1:91,2] = PR[GP1:90,2] + -35.703;
   1:L PR[91] 10mm/sec CNT100;
   1:  PR[GP1:91,1] = PR[GP1:90,1] + 25.702;
   1:  PR[GP1:91,2] = PR[GP1:90,2] + -36.102;
   1:L PR[91] 10mm/sec CNT100;
   1:  PR[GP1:91,1] = PR[GP1:90,1] + 27.081;
   1:  PR[GP1:91,2] = PR[GP1:90,2] + -36.151;
   1:L PR[91] 10mm/sec CNT100;
   1:  PR[GP1:91,1] = PR[GP1:90,1] + 32.618;
   1:  PR[GP1:91,2] = PR[GP1:90,2] + -35.536;
   1:L PR[91] 10mm/sec CNT100;
   1:  PR[GP1:91,1] = PR[GP1:90,1] + 33.028;
   1:  PR[GP1:91,2] = PR[GP1:90,2] + -35.427;
   1:L PR[91] 10mm/sec CNT100;
   1:  PR[GP1:91,1] = PR[GP1:90,1] + 37.436;
   1:  PR[GP1:91,2] = PR[GP1:90,2] + -33.723;
   1:L PR[91] 10mm/sec CNT100;
   1:  PR[GP1:91,1] = PR[GP1:90,1] + 37.766;
   1:  PR[GP1:91,2] = PR[GP1:90,2] + -33.571;
   1:L PR[91] 10mm/sec CNT100;
   1:  PR[GP1:91,1] = PR[GP1:90,1] + 37.979;
   1:  PR[GP1:91,2] = PR[GP1:90,2] + -33.419;
   1:L PR[91] 10mm/sec CNT100;
   1:  PR[GP1:91,1] = PR[GP1:90,1] + 41.444;
   1:  PR[GP1:91,2] = PR[GP1:90,2] + -30.698;
   1:L PR[91] 10mm/sec CNT100;
   1:  PR[GP1:91,1] = PR[GP1:90,1] + 41.594;
   1:  PR[GP1:91,2] = PR[GP1:90,2] + -30.538;
   1:L PR[91] 10mm/sec CNT100;
   1:  PR[GP1:91,1] = PR[GP1:90,1] + 43.787;
   1:  PR[GP1:91,2] = PR[GP1:90,2] + -27.268;
   1:L PR[91] 10mm/sec CNT100;
   1:  PR[GP1:91,1] = PR[GP1:90,1] + 43.900;
   1:  PR[GP1:91,2] = PR[GP1:90,2] + -27.079;
   1:L PR[91] 10mm/sec CNT100;
   1:  PR[GP1:91,1] = PR[GP1:90,1] + 44.954;
   1:  PR[GP1:91,2] = PR[GP1:90,2] + -23.856;
   1:L PR[91] 10mm/sec CNT100;
   1:  PR[GP1:91,1] = PR[GP1:90,1] + 45.253;
   1:  PR[GP1:91,2] = PR[GP1:90,2] + -20.854;
   1:L PR[91] 10mm/sec CNT100;
   1:  PR[GP1:91,1] = PR[GP1:90,1] + 45.231;
   1:  PR[GP1:91,2] = PR[GP1:90,2] + -20.499;
   1:L PR[91] 10mm/sec CNT100;
   1:  PR[GP1:91,1] = PR[GP1:90,1] + 45.005;
   1:  PR[GP1:91,2] = PR[GP1:90,2] + -17.852;
   1:L PR[91] 10mm/sec CNT100;
   1:  PR[GP1:91,1] = PR[GP1:90,1] + 44.272;
   1:  PR[GP1:91,2] = PR[GP1:90,2] + -14.875;
   1:L PR[91] 10mm/sec CNT100;
   1:  PR[GP1:91,1] = PR[GP1:90,1] + 43.161;
   1:  PR[GP1:91,2] = PR[GP1:90,2] + -12.090;
   1:L PR[91] 10mm/sec CNT100;
   1:  PR[GP1:91,1] = PR[GP1:90,1] + 41.716;
   1:  PR[GP1:91,2] = PR[GP1:90,2] + -9.444;
   1:L PR[91] 10mm/sec CNT100;
   1:  PR[GP1:91,1] = PR[GP1:90,1] + 40.781;
   1:  PR[GP1:91,2] = PR[GP1:90,2] + -8.090;
   1:L PR[91] 10mm/sec CNT100;
   1:  PR[GP1:91,1] = PR[GP1:90,1] + 39.109;
   1:  PR[GP1:91,2] = PR[GP1:90,2] + -5.931;
   1:L PR[91] 10mm/sec CNT100;
   1:  PR[GP1:91,1] = PR[GP1:90,1] + 37.856;
   1:  PR[GP1:91,2] = PR[GP1:90,2] + -4.598;
   1:L PR[91] 10mm/sec CNT100;
   1:  PR[GP1:91,1] = PR[GP1:90,1] + 35.494;
   1:  PR[GP1:91,2] = PR[GP1:90,2] + -2.519;
   1:L PR[91] 10mm/sec CNT100;
   1:  PR[GP1:91,1] = PR[GP1:90,1] + 32.551;
   1:  PR[GP1:91,2] = PR[GP1:90,2] + -0.388;
   1:L PR[91] 10mm/sec CNT100;
   1:  PR[GP1:91,1] = PR[GP1:90,1] + 30.080;
   1:  PR[GP1:91,2] = PR[GP1:90,2] + 1.054;
   1:L PR[91] 10mm/sec CNT100;
   1:  PR[GP1:91,1] = PR[GP1:90,1] + 29.130;
   1:  PR[GP1:91,2] = PR[GP1:90,2] + 1.568;
   1:L PR[91] 10mm/sec CNT100;
   1:  PR[GP1:91,1] = PR[GP1:90,1] + 27.148;
   1:  PR[GP1:91,2] = PR[GP1:90,2] + 2.485;
   1:L PR[91] 10mm/sec CNT100;
   1:  PR[GP1:91,1] = PR[GP1:90,1] + 25.363;
   1:  PR[GP1:91,2] = PR[GP1:90,2] + 3.126;
   1:L PR[91] 10mm/sec CNT100;
   1:  PR[GP1:91,1] = PR[GP1:90,1] + 24.181;
   1:  PR[GP1:91,2] = PR[GP1:90,2] + 3.607;
   1:L PR[91] 10mm/sec CNT100;
   1:  PR[GP1:91,1] = PR[GP1:90,1] + 22.716;
   1:  PR[GP1:91,2] = PR[GP1:90,2] + 4.045;
   1:L PR[91] 10mm/sec CNT100;
   1:  PR[GP1:91,1] = PR[GP1:90,1] + 20.918;
   1:  PR[GP1:91,2] = PR[GP1:90,2] + 4.485;
   1:L PR[91] 10mm/sec CNT100;
   1:  PR[GP1:91,1] = PR[GP1:90,1] + 20.299;
   1:  PR[GP1:91,2] = PR[GP1:90,2] + 4.602;
   1:L PR[91] 10mm/sec CNT100;
   1:  PR[GP1:91,1] = PR[GP1:90,1] + 20.125;
   1:  PR[GP1:91,2] = PR[GP1:90,2] + 4.654;
   1:L PR[91] 10mm/sec CNT100;
   1:  PR[GP1:91,1] = PR[GP1:90,1] + 18.327;
   1:  PR[GP1:91,2] = PR[GP1:90,2] + 4.929;
   1:L PR[91] 10mm/sec CNT100;
   1:  PR[GP1:91,1] = PR[GP1:90,1] + 17.294;
   1:  PR[GP1:91,2] = PR[GP1:90,2] + 5.041;
   1:L PR[91] 10mm/sec CNT100;
   1:  PR[GP1:91,1] = PR[GP1:90,1] + 14.652;
   1:  PR[GP1:91,2] = PR[GP1:90,2] + 5.152;
   1:L PR[91] 10mm/sec CNT100;
   1:  PR[GP1:91,1] = PR[GP1:90,1] + 13.670;
   1:  PR[GP1:91,2] = PR[GP1:90,2] + 5.116;
   1:L PR[91] 10mm/sec CNT100;
   1:  PR[GP1:91,1] = PR[GP1:90,1] + 11.603;
   1:  PR[GP1:91,2] = PR[GP1:90,2] + 4.983;
   1:L PR[91] 10mm/sec CNT100;
   1:  PR[GP1:91,1] = PR[GP1:90,1] + 9.273;
   1:  PR[GP1:91,2] = PR[GP1:90,2] + 4.525;
   1:L PR[91] 10mm/sec CNT100;
   1:  PR[GP1:91,1] = PR[GP1:90,1] + 8.260;
   1:  PR[GP1:91,2] = PR[GP1:90,2] + 4.344;
   1:L PR[91] 10mm/sec CNT100;
   1:  PR[GP1:91,1] = PR[GP1:90,1] + 7.357;
   1:  PR[GP1:91,2] = PR[GP1:90,2] + 4.067;
   1:L PR[91] 10mm/sec CNT100;
   1:  PR[GP1:91,1] = PR[GP1:90,1] + 6.676;
   1:  PR[GP1:91,2] = PR[GP1:90,2] + 3.770;
   1:L PR[91] 10mm/sec CNT100;
   1:  PR[GP1:91,1] = PR[GP1:90,1] + 4.484;
   1:  PR[GP1:91,2] = PR[GP1:90,2] + 2.910;
   1:L PR[91] 10mm/sec CNT100;
   1:  PR[GP1:91,1] = PR[GP1:90,1] + 4.060;
   1:  PR[GP1:91,2] = PR[GP1:90,2] + 2.690;
   1:L PR[91] 10mm/sec CNT100;
   1:  PR[GP1:91,1] = PR[GP1:90,1] + 1.817;
   1:  PR[GP1:91,2] = PR[GP1:90,2] + 1.258;
   1:L PR[91] 10mm/sec CNT100;
   1:  PR[GP1:91,1] = PR[GP1:90,1] + 0.148;
   1:  PR[GP1:91,2] = PR[GP1:90,2] + -0.210;
   1:L PR[91] 10mm/sec CNT100;
   1:  PR[GP1:91,1] = PR[GP1:90,1] + -0.116;
   1:  PR[GP1:91,2] = PR[GP1:90,2] + -0.495;
   1:L PR[91] 10mm/sec CNT100;
   1:  PR[GP1:91,1] = PR[GP1:90,1] + -1.468;
   1:  PR[GP1:91,2] = PR[GP1:90,2] + -2.163;
   1:L PR[91] 10mm/sec CNT100;
   1:  PR[GP1:91,1] = PR[GP1:90,1] + -2.498;
   1:  PR[GP1:91,2] = PR[GP1:90,2] + -4.004;
   1:L PR[91] 10mm/sec CNT100;
   1:  PR[GP1:91,1] = PR[GP1:90,1] + -2.685;
   1:  PR[GP1:91,2] = PR[GP1:90,2] + -4.360;
   1:L PR[91] 10mm/sec CNT100;
   1:  PR[GP1:91,1] = PR[GP1:90,1] + -3.376;
   1:  PR[GP1:91,2] = PR[GP1:90,2] + -6.287;
   1:L PR[91] 10mm/sec CNT100;
   1:  PR[GP1:91,1] = PR[GP1:90,1] + -3.467;
   1:  PR[GP1:91,2] = PR[GP1:90,2] + -6.679;
   1:L PR[91] 10mm/sec CNT100;
   1:  PR[GP1:91,1] = PR[GP1:90,1] + -3.842;
   1:  PR[GP1:91,2] = PR[GP1:90,2] + -8.716;
   1:L PR[91] 10mm/sec CNT100;
   1:  PR[GP1:91,1] = PR[GP1:90,1] + -3.882;
   1:  PR[GP1:91,2] = PR[GP1:90,2] + -10.815;
   1:L PR[91] 10mm/sec CNT100;
   1:  PR[GP1:91,1] = PR[GP1:90,1] + -3.862;
   1:  PR[GP1:91,2] = PR[GP1:90,2] + -11.203;
   1:L PR[91] 10mm/sec CNT100;
   1:  PR[GP1:91,1] = PR[GP1:90,1] + -3.824;
   1:  PR[GP1:91,2] = PR[GP1:90,2] + -11.437;
   1:L PR[91] 10mm/sec CNT100;
   1:  PR[GP1:91,1] = PR[GP1:90,1] + -3.544;
   1:  PR[GP1:91,2] = PR[GP1:90,2] + -13.362;
   1:L PR[91] 10mm/sec CNT100;
   1:  PR[GP1:91,1] = PR[GP1:90,1] + -3.316;
   1:  PR[GP1:91,2] = PR[GP1:90,2] + -14.057;
   1:L PR[91] 10mm/sec CNT100;
   1:  PR[GP1:91,1] = PR[GP1:90,1] + -2.515;
   1:  PR[GP1:91,2] = PR[GP1:90,2] + -16.701;
   1:L PR[91] 10mm/sec CNT100;
   1:  PR[GP1:91,1] = PR[GP1:90,1] + -1.373;
   1:  PR[GP1:91,2] = PR[GP1:90,2] + -19.154;
   1:L PR[91] 10mm/sec CNT100;
   1:  PR[GP1:91,1] = PR[GP1:90,1] + -1.069;
   1:  PR[GP1:91,2] = PR[GP1:90,2] + -19.664;
   1:L PR[91] 10mm/sec CNT100;
   1:  PR[GP1:91,1] = PR[GP1:90,1] + 2.304;
   1:  PR[GP1:91,2] = PR[GP1:90,2] + -24.337;
   1:L PR[91] 10mm/sec CNT100;
   1:  PR[GP1:91,1] = PR[GP1:90,1] + 4.017;
   1:  PR[GP1:91,2] = PR[GP1:90,2] + -26.127;
   1:L PR[91] 10mm/sec CNT100;
   1:  PR[GP1:91,1] = PR[GP1:90,1] + 5.297;
   1:  PR[GP1:91,2] = PR[GP1:90,2] + -27.128;
   1:L PR[91] 10mm/sec CNT100;
   1:  PR[GP1:91,1] = PR[GP1:90,1] + 7.670;
   1:  PR[GP1:91,2] = PR[GP1:90,2] + -29.157;
   1:L PR[91] 10mm/sec CNT100;
   1:  PR[GP1:91,1] = PR[GP1:90,1] + 11.968;
   1:  PR[GP1:91,2] = PR[GP1:90,2] + -31.818;
   1:L PR[91] 10mm/sec CNT100;
   1:  PR[GP1:91,1] = PR[GP1:90,1] + 13.448;
   1:  PR[GP1:91,2] = PR[GP1:90,2] + -32.684;
   1:L PR[91] 10mm/sec CNT100;
   1:  PR[GP1:91,1] = PR[GP1:90,1] + 20.392;
   1:  PR[GP1:91,2] = PR[GP1:90,2] + -35.346;
   1:L PR[91] 10mm/sec CNT100;
   1:  PR[GP1:91,1] = PR[GP1:90,1] + 22.229;
   1:  PR[GP1:91,2] = PR[GP1:90,2] + -35.703;
   1:L PR[91] 10mm/sec CNT100;
   1:  PR[GP1:91,1] = PR[GP1:90,1] + 25.702;
   1:  PR[GP1:91,2] = PR[GP1:90,2] + -36.102;
   1:L PR[91] 10mm/sec CNT100;
   1:  PR[GP1:91,1] = PR[GP1:90,1] + 27.081;
   1:  PR[GP1:91,2] = PR[GP1:90,2] + -36.151;
   1:L PR[91] 10mm/sec CNT100;
   1:  PR[GP1:91,1] = PR[GP1:90,1] + 32.618;
   1:  PR[GP1:91,2] = PR[GP1:90,2] + -35.536;
   1:L PR[91] 10mm/sec CNT100;
   1:  PR[GP1:91,1] = PR[GP1:90,1] + 33.028;
   1:  PR[GP1:91,2] = PR[GP1:90,2] + -35.427;
   1:L PR[91] 10mm/sec CNT100;
   1:  PR[GP1:91,1] = PR[GP1:90,1] + 37.436;
   1:  PR[GP1:91,2] = PR[GP1:90,2] + -33.723;
   1:L PR[91] 10mm/sec CNT100;
   1:  PR[GP1:91,1] = PR[GP1:90,1] + 37.766;
   1:  PR[GP1:91,2] = PR[GP1:90,2] + -33.571;
   1:L PR[91] 10mm/sec CNT100;
   1:  PR[GP1:91,1] = PR[GP1:90,1] + 37.979;
   1:  PR[GP1:91,2] = PR[GP1:90,2] + -33.419;
   1:L PR[91] 10mm/sec CNT100;
   1:  PR[GP1:91,1] = PR[GP1:90,1] + 41.444;
   1:  PR[GP1:91,2] = PR[GP1:90,2] + -30.698;
   1:L PR[91] 10mm/sec CNT100;
   1:  PR[GP1:91,1] = PR[GP1:90,1] + 41.594;
   1:  PR[GP1:91,2] = PR[GP1:90,2] + -30.538;
   1:L PR[91] 10mm/sec CNT100;
   1:  PR[GP1:91,1] = PR[GP1:90,1] + 43.787;
   1:  PR[GP1:91,2] = PR[GP1:90,2] + -27.268;
   1:L PR[91] 10mm/sec CNT100;
   1:  PR[GP1:91,1] = PR[GP1:90,1] + 43.900;
   1:  PR[GP1:91,2] = PR[GP1:90,2] + -27.079;
   1:L PR[91] 10mm/sec CNT100;
   1:  PR[GP1:91,1] = PR[GP1:90,1] + 44.954;
   1:  PR[GP1:91,2] = PR[GP1:90,2] + -23.856;
   1:L PR[91] 10mm/sec CNT100;
   1:  PR[GP1:91,1] = PR[GP1:90,1] + 45.253;
   1:  PR[GP1:91,2] = PR[GP1:90,2] + -20.854;
   1:L PR[91] 10mm/sec CNT100;
   1:  PR[GP1:91,1] = PR[GP1:90,1] + 45.231;
   1:  PR[GP1:91,2] = PR[GP1:90,2] + -20.499;
   1:L PR[91] 10mm/sec CNT100;
   1:  PR[GP1:91,1] = PR[GP1:90,1] + 45.005;
   1:  PR[GP1:91,2] = PR[GP1:90,2] + -17.852;
   1:L PR[91] 10mm/sec CNT100;
   1:  PR[GP1:91,1] = PR[GP1:90,1] + 44.272;
   1:  PR[GP1:91,2] = PR[GP1:90,2] + -14.875;
   1:L PR[91] 10mm/sec CNT100;
   1:  PR[GP1:91,1] = PR[GP1:90,1] + 43.161;
   1:  PR[GP1:91,2] = PR[GP1:90,2] + -12.090;
   1:L PR[91] 10mm/sec CNT100;
   1:  PR[GP1:91,1] = PR[GP1:90,1] + 41.716;
   1:  PR[GP1:91,2] = PR[GP1:90,2] + -9.444;
   1:L PR[91] 10mm/sec CNT100;
   1:  PR[GP1:91,1] = PR[GP1:90,1] + 40.781;
   1:  PR[GP1:91,2] = PR[GP1:90,2] + -8.090;
   1:L PR[91] 10mm/sec CNT100;
   1:  PR[GP1:91,1] = PR[GP1:90,1] + 39.109;
   1:  PR[GP1:91,2] = PR[GP1:90,2] + -5.931;
   1:L PR[91] 10mm/sec CNT100;
   1:  PR[GP1:91,1] = PR[GP1:90,1] + 37.856;
   1:  PR[GP1:91,2] = PR[GP1:90,2] + -4.598;
   1:L PR[91] 10mm/sec CNT100;
   1:  PR[GP1:91,1] = PR[GP1:90,1] + 35.494;
   1:  PR[GP1:91,2] = PR[GP1:90,2] + -2.519;
   1:L PR[91] 10mm/sec CNT100;
   1:  PR[GP1:91,1] = PR[GP1:90,1] + 32.551;
   1:  PR[GP1:91,2] = PR[GP1:90,2] + -0.388;
   1:L PR[91] 10mm/sec CNT100;
   1:  PR[GP1:91,1] = PR[GP1:90,1] + 30.080;
   1:  PR[GP1:91,2] = PR[GP1:90,2] + 1.054;
   1:L PR[91] 10mm/sec CNT100;
   1:  PR[GP1:91,1] = PR[GP1:90,1] + 29.130;
   1:  PR[GP1:91,2] = PR[GP1:90,2] + 1.568;
   1:L PR[91] 10mm/sec CNT100;
   1:  PR[GP1:91,1] = PR[GP1:90,1] + 27.148;
   1:  PR[GP1:91,2] = PR[GP1:90,2] + 2.485;
   1:L PR[91] 10mm/sec CNT100;
   1:  PR[GP1:91,1] = PR[GP1:90,1] + 25.363;
   1:  PR[GP1:91,2] = PR[GP1:90,2] + 3.126;
   1:L PR[91] 10mm/sec CNT100;
   1:  PR[GP1:91,1] = PR[GP1:90,1] + 24.181;
   1:  PR[GP1:91,2] = PR[GP1:90,2] + 3.607;
   1:L PR[91] 10mm/sec CNT100;
   1:  PR[GP1:91,1] = PR[GP1:90,1] + 22.716;
   1:  PR[GP1:91,2] = PR[GP1:90,2] + 4.045;
   1:L PR[91] 10mm/sec CNT100;
   1:  PR[GP1:91,1] = PR[GP1:90,1] + 20.918;
   1:  PR[GP1:91,2] = PR[GP1:90,2] + 4.485;
   1:L PR[91] 10mm/sec CNT100;
   1:  PR[GP1:91,1] = PR[GP1:90,1] + 20.299;
   1:  PR[GP1:91,2] = PR[GP1:90,2] + 4.602;
   1:L PR[91] 10mm/sec CNT100;
   1:  PR[GP1:91,1] = PR[GP1:90,1] + 20.125;
   1:  PR[GP1:91,2] = PR[GP1:90,2] + 4.654;
   1:L PR[91] 10mm/sec CNT100;
   1:  PR[GP1:91,1] = PR[GP1:90,1] + 18.327;
   1:  PR[GP1:91,2] = PR[GP1:90,2] + 4.929;
   1:L PR[91] 10mm/sec CNT100;
   1:  PR[GP1:91,1] = PR[GP1:90,1] + 17.294;
   1:  PR[GP1:91,2] = PR[GP1:90,2] + 5.041;
   1:L PR[91] 10mm/sec CNT100;
   1:  PR[GP1:91,1] = PR[GP1:90,1] + 14.652;
   1:  PR[GP1:91,2] = PR[GP1:90,2] + 5.152;
   1:L PR[91] 10mm/sec CNT100;
   1:  PR[GP1:91,1] = PR[GP1:90,1] + 13.670;
   1:  PR[GP1:91,2] = PR[GP1:90,2] + 5.116;
   1:L PR[91] 10mm/sec CNT100;
   1:  PR[GP1:91,1] = PR[GP1:90,1] + 11.603;
   1:  PR[GP1:91,2] = PR[GP1:90,2] + 4.983;
   1:L PR[91] 10mm/sec CNT100;
   1:  PR[GP1:91,1] = PR[GP1:90,1] + 9.273;
   1:  PR[GP1:91,2] = PR[GP1:90,2] + 4.525;
   1:L PR[91] 10mm/sec CNT100;
   1:  PR[GP1:91,1] = PR[GP1:90,1] + 8.260;
   1:  PR[GP1:91,2] = PR[GP1:90,2] + 4.344;
   1:L PR[91] 10mm/sec CNT100;
   1:  PR[GP1:91,1] = PR[GP1:90,1] + 7.357;
   1:  PR[GP1:91,2] = PR[GP1:90,2] + 4.067;
   1:L PR[91] 10mm/sec CNT100;
   1:  PR[GP1:91,1] = PR[GP1:90,1] + 6.676;
   1:  PR[GP1:91,2] = PR[GP1:90,2] + 3.770;
   1:L PR[91] 10mm/sec CNT100;
   1:  PR[GP1:91,1] = PR[GP1:90,1] + 4.484;
   1:  PR[GP1:91,2] = PR[GP1:90,2] + 2.910;
   1:L PR[91] 10mm/sec CNT100;
   1:  PR[GP1:91,1] = PR[GP1:90,1] + 4.060;
   1:  PR[GP1:91,2] = PR[GP1:90,2] + 2.690;
   1:L PR[91] 10mm/sec CNT100;
   1:  PR[GP1:91,1] = PR[GP1:90,1] + 1.817;
   1:  PR[GP1:91,2] = PR[GP1:90,2] + 1.258;
   1:L PR[91] 10mm/sec CNT100;
   1:  PR[GP1:91,1] = PR[GP1:90,1] + 0.148;
   1:  PR[GP1:91,2] = PR[GP1:90,2] + -0.210;
   1:L PR[91] 10mm/sec CNT100;
   1:  PR[GP1:91,1] = PR[GP1:90,1] + -0.116;
   1:  PR[GP1:91,2] = PR[GP1:90,2] + -0.495;
   1:L PR[91] 10mm/sec CNT100;
   1:  PR[GP1:91,1] = PR[GP1:90,1] + -1.468;
   1:  PR[GP1:91,2] = PR[GP1:90,2] + -2.163;
   1:L PR[91] 10mm/sec CNT100;
   1:  PR[GP1:91,1] = PR[GP1:90,1] + -2.498;
   1:  PR[GP1:91,2] = PR[GP1:90,2] + -4.004;
   1:L PR[91] 10mm/sec CNT100;
   1:  PR[GP1:91,1] = PR[GP1:90,1] + -2.685;
   1:  PR[GP1:91,2] = PR[GP1:90,2] + -4.360;
   1:L PR[91] 10mm/sec CNT100;
   1:  PR[GP1:91,1] = PR[GP1:90,1] + -3.376;
   1:  PR[GP1:91,2] = PR[GP1:90,2] + -6.287;
   1:L PR[91] 10mm/sec CNT100;
   1:  PR[GP1:91,1] = PR[GP1:90,1] + -3.467;
   1:  PR[GP1:91,2] = PR[GP1:90,2] + -6.679;
   1:L PR[91] 10mm/sec CNT100;
   1:  PR[GP1:91,1] = PR[GP1:90,1] + -3.842;
   1:  PR[GP1:91,2] = PR[GP1:90,2] + -8.716;
   1:L PR[91] 10mm/sec CNT100;
   1:  PR[GP1:91,1] = PR[GP1:90,1] + -3.882;
   1:  PR[GP1:91,2] = PR[GP1:90,2] + -10.815;
   1:L PR[91] 10mm/sec CNT100;
   1:  PR[GP1:91,1] = PR[GP1:90,1] + -3.862;
   1:  PR[GP1:91,2] = PR[GP1:90,2] + -11.203;
   1:L PR[91] 10mm/sec CNT100;
   1:  PR[GP1:91,1] = PR[GP1:90,1] + -3.824;
   1:  PR[GP1:91,2] = PR[GP1:90,2] + -11.437;
   1:L PR[91] 10mm/sec CNT100;
   1:  PR[GP1:91,1] = PR[GP1:90,1] + -3.544;
   1:  PR[GP1:91,2] = PR[GP1:90,2] + -13.362;
   1:L PR[91] 10mm/sec CNT100;
   1:  PR[GP1:91,1] = PR[GP1:90,1] + -3.316;
   1:  PR[GP1:91,2] = PR[GP1:90,2] + -14.057;
   1:L PR[91] 10mm/sec CNT100;
   1:  CALL HOME_ALL;
/POS
/END
